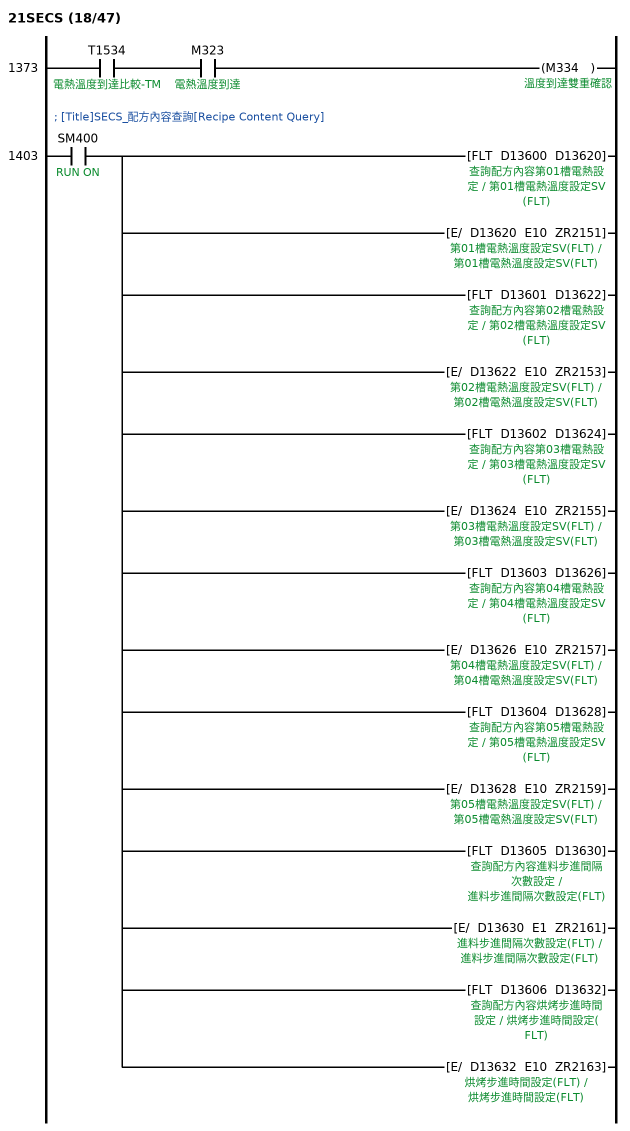
[picture p96: ladder of 21SECS, rungs at steps 1373 to 1403]
1373  LD      T1534  ; 電熱溫度到達比較-TM
      AND     M323  ; 電熱溫度到達
      OUT     M334  ; 溫度到達雙重確認
; [Title]SECS_配方內容查詢[Recipe Content Query]
1403  LD      SM400  ; RUN ON
      FLT     D13600 D13620  ; 查詢配方內容第01槽電熱設定 / 第01槽電熱溫度設定SV(FLT)
      E/      D13620 E10 ZR2151  ; 第01槽電熱溫度設定SV(FLT)
      FLT     D13601 D13622  ; 查詢配方內容第02槽電熱設定 / 第02槽電熱溫度設定SV(FLT)
      E/      D13622 E10 ZR2153  ; 第02槽電熱溫度設定SV(FLT)
      FLT     D13602 D13624  ; 查詢配方內容第03槽電熱設定 / 第03槽電熱溫度設定SV(FLT)
      E/      D13624 E10 ZR2155  ; 第03槽電熱溫度設定SV(FLT)
      FLT     D13603 D13626  ; 查詢配方內容第04槽電熱設定 / 第04槽電熱溫度設定SV(FLT)
      E/      D13626 E10 ZR2157  ; 第04槽電熱溫度設定SV(FLT)
      FLT     D13604 D13628  ; 查詢配方內容第05槽電熱設定 / 第05槽電熱溫度設定SV(FLT)
      E/      D13628 E10 ZR2159  ; 第05槽電熱溫度設定SV(FLT)
      FLT     D13605 D13630  ; 查詢配方內容進料步進間隔次數設定 / 進料步進間隔次數設定(FLT)
      E/      D13630 E1 ZR2161  ; 進料步進間隔次數設定(FLT)
      FLT     D13606 D13632  ; 查詢配方內容烘烤步進時間設定 / 烘烤步進時間設定(FLT)
      E/      D13632 E10 ZR2163  ; 烘烤步進時間設定(FLT)
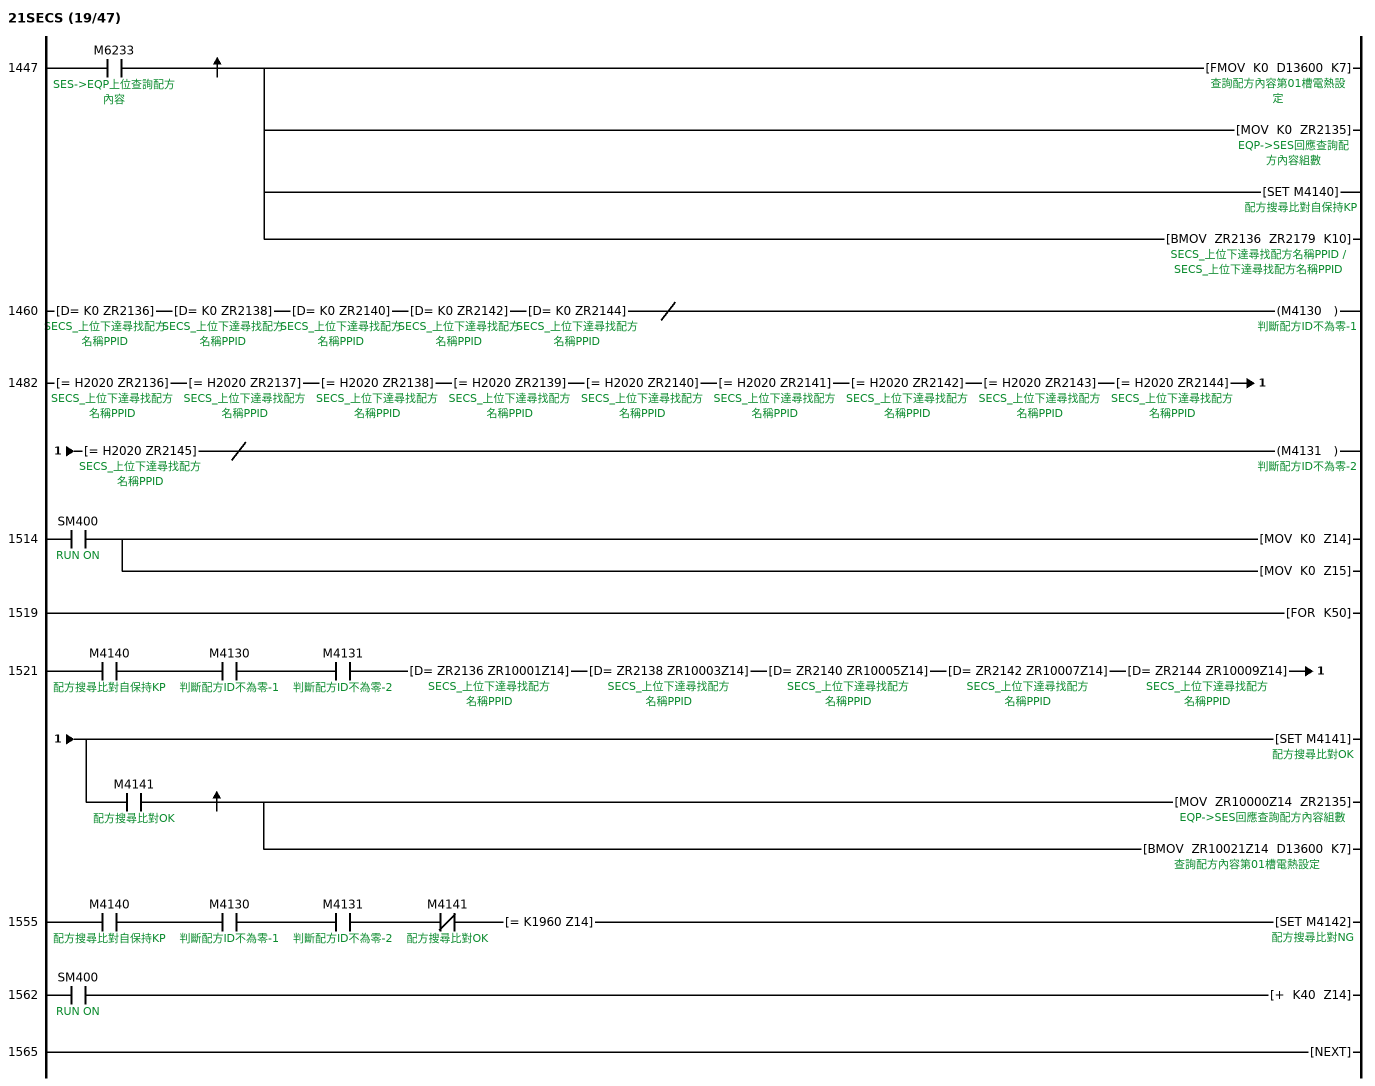
1447  LD      M6233  ; SES->EQP上位查詢配方內容
      MEP
      FMOV    K0 D13600 K7
      MOV     K0 ZR2135  ; EQP->SES回應查詢配方內容組數
      SET     M4140  ; 配方搜尋比對自保持KP
      BMOV    ZR2136 ZR2179 K10  ; SECS_上位下達尋找配方名稱PPID / SECS_上位下達尋找配方名稱PPID
1460  LDD=    K0 ZR2136  ; SECS_上位下達尋找配方名稱PPID
      ANDD=   K0 ZR2138  ; SECS_上位下達尋找配方名稱PPID
      ANDD=   K0 ZR2140  ; SECS_上位下達尋找配方名稱PPID
      ANDD=   K0 ZR2142  ; SECS_上位下達尋找配方名稱PPID
      ANDD=   K0 ZR2144  ; SECS_上位下達尋找配方名稱PPID
      INV
      OUT     M4130  ; 判斷配方ID不為零-1
1482  LD=     H2020 ZR2136  ; SECS_上位下達尋找配方名稱PPID
      AND=    H2020 ZR2137  ; SECS_上位下達尋找配方名稱PPID
      AND=    H2020 ZR2138  ; SECS_上位下達尋找配方名稱PPID
      AND=    H2020 ZR2139  ; SECS_上位下達尋找配方名稱PPID
      AND=    H2020 ZR2140  ; SECS_上位下達尋找配方名稱PPID
      AND=    H2020 ZR2141  ; SECS_上位下達尋找配方名稱PPID
      AND=    H2020 ZR2142  ; SECS_上位下達尋找配方名稱PPID
      AND=    H2020 ZR2143  ; SECS_上位下達尋找配方名稱PPID
      AND=    H2020 ZR2144  ; SECS_上位下達尋找配方名稱PPID
      AND=    H2020 ZR2145  ; SECS_上位下達尋找配方名稱PPID
      INV
      OUT     M4131  ; 判斷配方ID不為零-2
1514  LD      SM400  ; RUN ON
      MOV     K0 Z14
      MOV     K0 Z15
1519  FOR     K50
1521  LD      M4140  ; 配方搜尋比對自保持KP
      AND     M4130  ; 判斷配方ID不為零-1
      AND     M4131  ; 判斷配方ID不為零-2
      ANDD=   ZR2136 ZR10001Z14  ; SECS_上位下達尋找配方名稱PPID
      ANDD=   ZR2138 ZR10003Z14  ; SECS_上位下達尋找配方名稱PPID
      ANDD=   ZR2140 ZR10005Z14  ; SECS_上位下達尋找配方名稱PPID
      ANDD=   ZR2142 ZR10007Z14  ; SECS_上位下達尋找配方名稱PPID
      ANDD=   ZR2144 ZR10009Z14  ; SECS_上位下達尋找配方名稱PPID
      SET     M4141  ; 配方搜尋比對OK
      AND     M4141  ; 配方搜尋比對OK
      MEP
      MOV     ZR10000Z14 ZR2135
      BMOV    ZR10021Z14 D13600 K7
1555  LD      M4140  ; 配方搜尋比對自保持KP
      AND     M4130  ; 判斷配方ID不為零-1
      AND     M4131  ; 判斷配方ID不為零-2
      ANI     M4141  ; 配方搜尋比對OK
      AND=    K1960 Z14
      SET     M4142  ; 配方搜尋比對NG
1562  LD      SM400  ; RUN ON
      +       K40 Z14
1565  NEXT
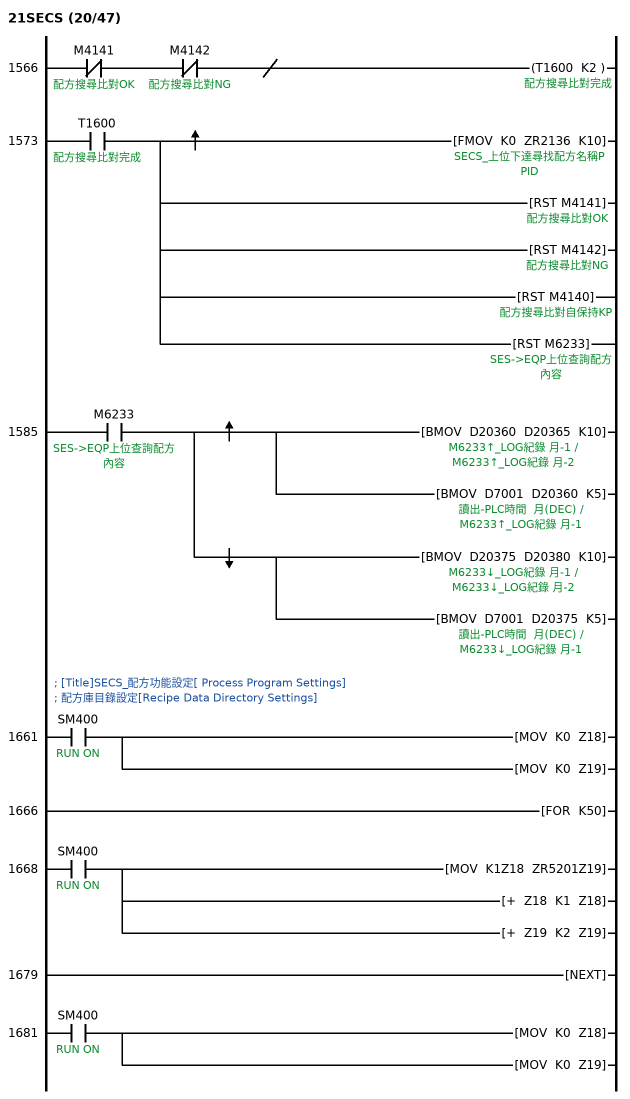
1566  LDI     M4141  ; 配方搜尋比對OK
      ANI     M4142  ; 配方搜尋比對NG
      INV
      OUT     T1600 K2  ; 配方搜尋比對完成
1573  LD      T1600  ; 配方搜尋比對完成
      MPS
      MEP
      FMOV    K0 ZR2136 K10
      MPP
      RST     M4141  ; 配方搜尋比對OK
      RST     M4142  ; 配方搜尋比對NG
      RST     M4140  ; 配方搜尋比對自保持KP
      RST     M6233  ; SES->EQP上位查詢配方內容
1585  LD      M6233  ; SES->EQP上位查詢配方內容
      MPS
      MEP
      BMOV    D20360 D20365 K10  ; M6233↑_LOG紀錄 月-1 / M6233↑_LOG紀錄 月-2
      BMOV    D7001 D20360 K5
      MPP
      MEF
      BMOV    D20375 D20380 K10  ; M6233↓_LOG紀錄 月-1 / M6233↓_LOG紀錄 月-2
      BMOV    D7001 D20375 K5
; [Title]SECS_配方功能設定[ Process Program Settings]
; 配方庫目錄設定[Recipe Data Directory Settings]
1661  LD      SM400  ; RUN ON
      MOV     K0 Z18
      MOV     K0 Z19
1666  FOR     K50
1668  LD      SM400  ; RUN ON
      MOV     K1Z18 ZR5201Z19
      +       Z18 K1 Z18
      +       Z19 K2 Z19
1679  NEXT
1681  LD      SM400  ; RUN ON
      MOV     K0 Z18
      MOV     K0 Z19
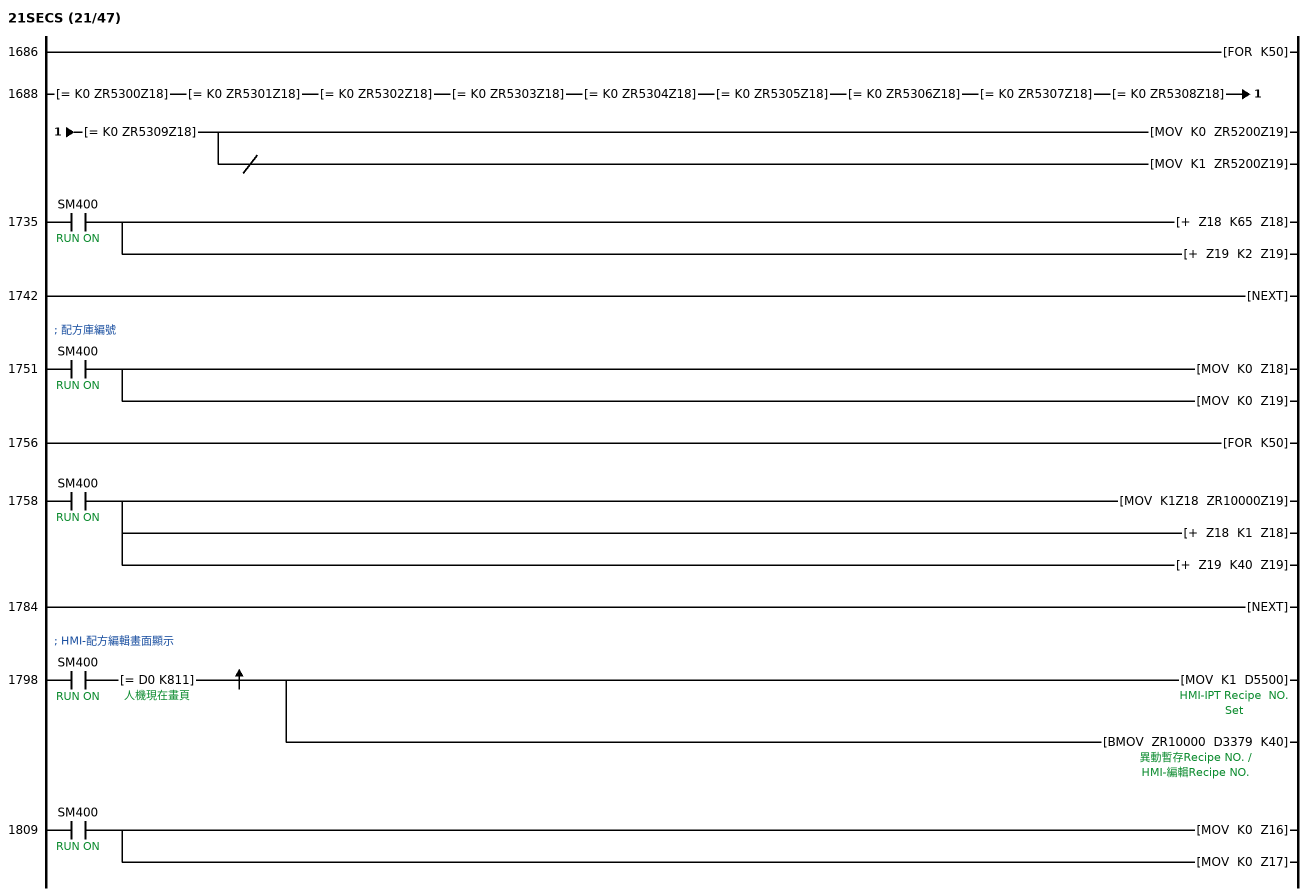
1686  FOR     K50
1688  LD=     K0 ZR5300Z18
      AND=    K0 ZR5301Z18
      AND=    K0 ZR5302Z18
      AND=    K0 ZR5303Z18
      AND=    K0 ZR5304Z18
      AND=    K0 ZR5305Z18
      AND=    K0 ZR5306Z18
      AND=    K0 ZR5307Z18
      AND=    K0 ZR5308Z18
      AND=    K0 ZR5309Z18
      MOV     K0 ZR5200Z19
      INV
      MOV     K1 ZR5200Z19
1735  LD      SM400  ; RUN ON
      +       Z18 K65 Z18
      +       Z19 K2 Z19
1742  NEXT
; 配方庫編號
1751  LD      SM400  ; RUN ON
      MOV     K0 Z18
      MOV     K0 Z19
1756  FOR     K50
1758  LD      SM400  ; RUN ON
      MOV     K1Z18 ZR10000Z19
        [note] 寫入配方參數Recipe NO.編號
      +       Z18 K1 Z18
      +       Z19 K40 Z19
1784  NEXT
; HMI-配方編輯畫面顯示
1798  LD      SM400  ; RUN ON
      AND=    D0 K811  ; 人機現在畫頁
      MEP
      MOV     K1 D5500  ; HMI-IPT Recipe  NO. Set
      BMOV    ZR10000 D3379 K40  ; 異動暫存Recipe NO. / HMI-編輯Recipe NO.
1809  LD      SM400  ; RUN ON
      MOV     K0 Z16
      MOV     K0 Z17
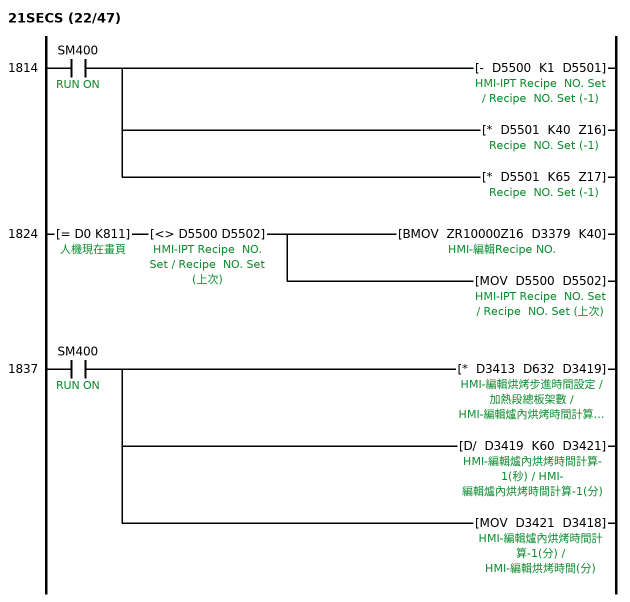
1814  LD      SM400  ; RUN ON
      -       D5500 K1 D5501  ; Recipe  NO. Set (-1)
      *       D5501 K40 Z16
      *       D5501 K65 Z17
1824  LD=     D0 K811  ; 人機現在畫頁
      AND<>   D5500 D5502  ; HMI-IPT Recipe  NO. Set / Recipe  NO. Set (上次)
      BMOV    ZR10000Z16 D3379 K40
      MOV     D5500 D5502
1837  LD      SM400  ; RUN ON
      *       D3413 D632 D3419  ; HMI-編輯烘烤步進時間設定 / 加熱段總板架數 / HMI-編輯爐內烘烤時間計算-1(秒)
        [note] 顯示輸入的秒數換算烘烤時間設定
      D/      D3419 K60 D3421  ; HMI-編輯爐內烘烤時間計算-1(分)
      MOV     D3421 D3418  ; HMI-編輯烘烤時間(分)
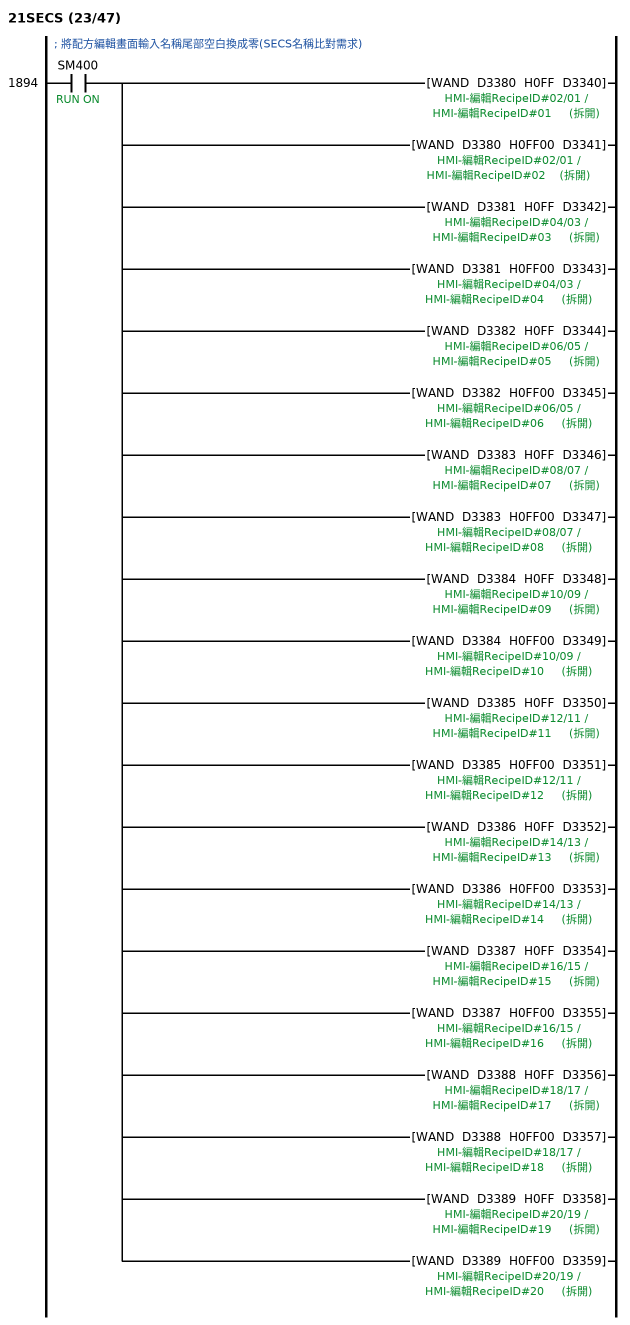
; 將配方編輯畫面輸入名稱尾部空白換成零(SECS名稱比對需求)
1894  LD      SM400  ; RUN ON
      WAND    D3380 H0FF D3340  ; HMI-編輯RecipeID#02/01 / HMI-編輯RecipeID#01     (拆開)
      WAND    D3380 H0FF00 D3341  ; HMI-編輯RecipeID#02    (拆開)
      WAND    D3381 H0FF D3342  ; HMI-編輯RecipeID#04/03 / HMI-編輯RecipeID#03     (拆開)
      WAND    D3381 H0FF00 D3343  ; HMI-編輯RecipeID#04     (拆開)
      WAND    D3382 H0FF D3344  ; HMI-編輯RecipeID#06/05 / HMI-編輯RecipeID#05     (拆開)
      WAND    D3382 H0FF00 D3345  ; HMI-編輯RecipeID#06     (拆開)
      WAND    D3383 H0FF D3346  ; HMI-編輯RecipeID#08/07 / HMI-編輯RecipeID#07     (拆開)
      WAND    D3383 H0FF00 D3347  ; HMI-編輯RecipeID#08     (拆開)
      WAND    D3384 H0FF D3348  ; HMI-編輯RecipeID#10/09 / HMI-編輯RecipeID#09     (拆開)
      WAND    D3384 H0FF00 D3349  ; HMI-編輯RecipeID#10     (拆開)
      WAND    D3385 H0FF D3350  ; HMI-編輯RecipeID#12/11 / HMI-編輯RecipeID#11     (拆開)
      WAND    D3385 H0FF00 D3351  ; HMI-編輯RecipeID#12     (拆開)
      WAND    D3386 H0FF D3352  ; HMI-編輯RecipeID#14/13 / HMI-編輯RecipeID#13     (拆開)
      WAND    D3386 H0FF00 D3353  ; HMI-編輯RecipeID#14     (拆開)
      WAND    D3387 H0FF D3354  ; HMI-編輯RecipeID#16/15 / HMI-編輯RecipeID#15     (拆開)
      WAND    D3387 H0FF00 D3355  ; HMI-編輯RecipeID#16     (拆開)
      WAND    D3388 H0FF D3356  ; HMI-編輯RecipeID#18/17 / HMI-編輯RecipeID#17     (拆開)
      WAND    D3388 H0FF00 D3357  ; HMI-編輯RecipeID#18     (拆開)
      WAND    D3389 H0FF D3358  ; HMI-編輯RecipeID#20/19 / HMI-編輯RecipeID#19     (拆開)
      WAND    D3389 H0FF00 D3359  ; HMI-編輯RecipeID#20     (拆開)
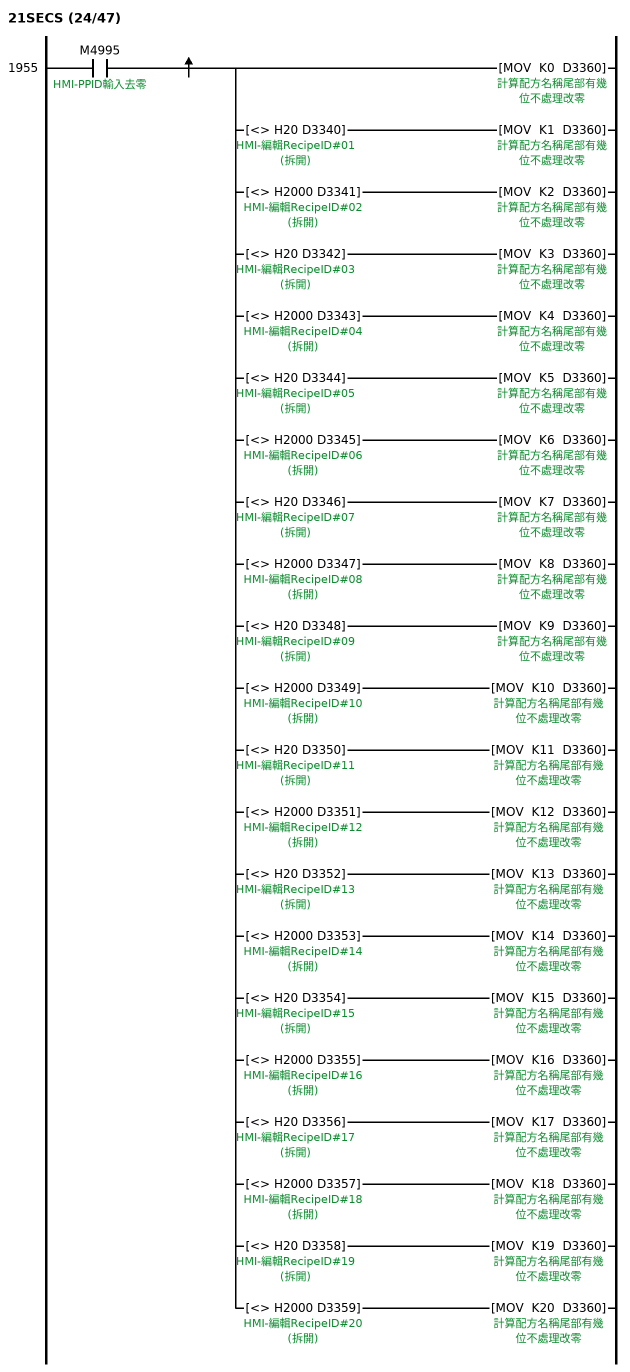
1955  LD      M4995  ; HMI-PPID輸入去零
      MEP
      MOV     K0 D3360  ; 計算配方名稱尾部有幾位不處理改零
      MPS
      AND<>   H20 D3340  ; HMI-編輯RecipeID#01     (拆開)
      MOV     K1 D3360
      MRD
      AND<>   H2000 D3341  ; HMI-編輯RecipeID#02    (拆開)
      MOV     K2 D3360
      MRD
      AND<>   H20 D3342  ; HMI-編輯RecipeID#03     (拆開)
      MOV     K3 D3360
      MRD
      AND<>   H2000 D3343  ; HMI-編輯RecipeID#04     (拆開)
      MOV     K4 D3360
      MRD
      AND<>   H20 D3344  ; HMI-編輯RecipeID#05     (拆開)
      MOV     K5 D3360
      MRD
      AND<>   H2000 D3345  ; HMI-編輯RecipeID#06     (拆開)
      MOV     K6 D3360
      MRD
      AND<>   H20 D3346  ; HMI-編輯RecipeID#07     (拆開)
      MOV     K7 D3360
      MRD
      AND<>   H2000 D3347  ; HMI-編輯RecipeID#08     (拆開)
      MOV     K8 D3360
      MRD
      AND<>   H20 D3348  ; HMI-編輯RecipeID#09     (拆開)
      MOV     K9 D3360
      MRD
      AND<>   H2000 D3349  ; HMI-編輯RecipeID#10     (拆開)
      MOV     K10 D3360
      MRD
      AND<>   H20 D3350  ; HMI-編輯RecipeID#11     (拆開)
      MOV     K11 D3360
      MRD
      AND<>   H2000 D3351  ; HMI-編輯RecipeID#12     (拆開)
      MOV     K12 D3360
      MRD
      AND<>   H20 D3352  ; HMI-編輯RecipeID#13     (拆開)
      MOV     K13 D3360
      MRD
      AND<>   H2000 D3353  ; HMI-編輯RecipeID#14     (拆開)
      MOV     K14 D3360
      MRD
      AND<>   H20 D3354  ; HMI-編輯RecipeID#15     (拆開)
      MOV     K15 D3360
      MRD
      AND<>   H2000 D3355  ; HMI-編輯RecipeID#16     (拆開)
      MOV     K16 D3360
      MRD
      AND<>   H20 D3356  ; HMI-編輯RecipeID#17     (拆開)
      MOV     K17 D3360
      MRD
      AND<>   H2000 D3357  ; HMI-編輯RecipeID#18     (拆開)
      MOV     K18 D3360
      MRD
      AND<>   H20 D3358  ; HMI-編輯RecipeID#19     (拆開)
      MOV     K19 D3360
      MPP
      AND<>   H2000 D3359  ; HMI-編輯RecipeID#20     (拆開)
      MOV     K20 D3360
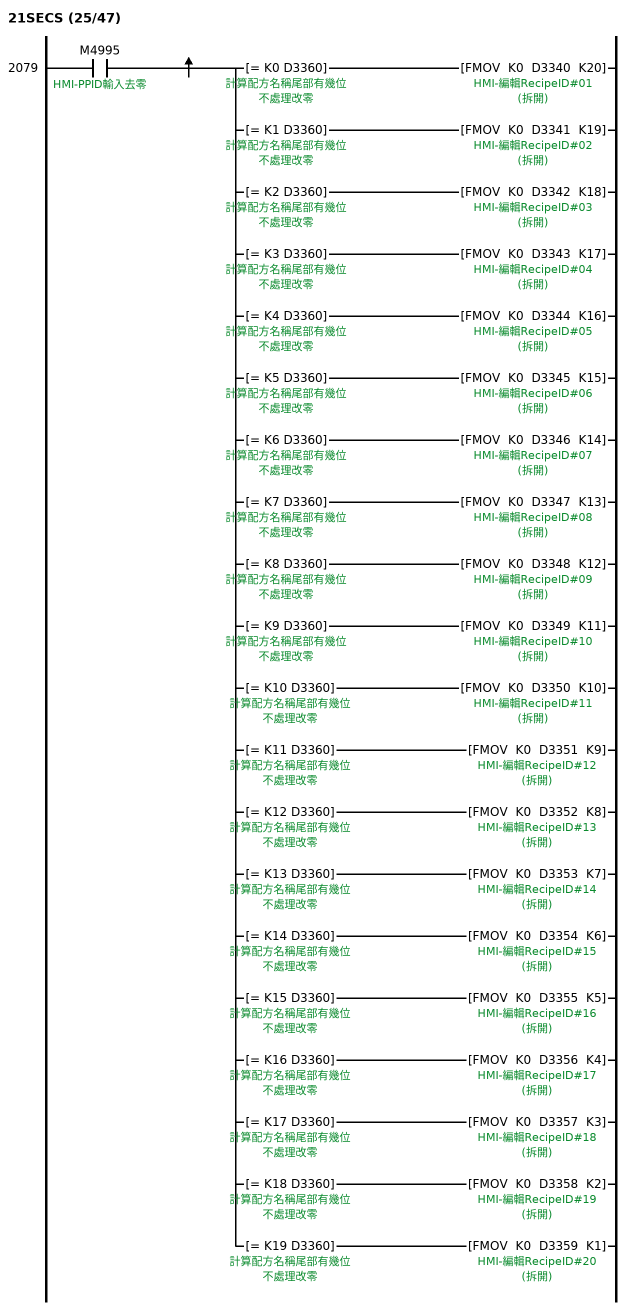
2079  LD      M4995  ; HMI-PPID輸入去零
      MEP
      MPS
      AND=    K0 D3360  ; 計算配方名稱尾部有幾位不處理改零
      FMOV    K0 D3340 K20
      MRD
      AND=    K1 D3360  ; 計算配方名稱尾部有幾位不處理改零
      FMOV    K0 D3341 K19
      MRD
      AND=    K2 D3360  ; 計算配方名稱尾部有幾位不處理改零
      FMOV    K0 D3342 K18
      MRD
      AND=    K3 D3360  ; 計算配方名稱尾部有幾位不處理改零
      FMOV    K0 D3343 K17
      MRD
      AND=    K4 D3360  ; 計算配方名稱尾部有幾位不處理改零
      FMOV    K0 D3344 K16
      MRD
      AND=    K5 D3360  ; 計算配方名稱尾部有幾位不處理改零
      FMOV    K0 D3345 K15
      MRD
      AND=    K6 D3360  ; 計算配方名稱尾部有幾位不處理改零
      FMOV    K0 D3346 K14
      MRD
      AND=    K7 D3360  ; 計算配方名稱尾部有幾位不處理改零
      FMOV    K0 D3347 K13
      MRD
      AND=    K8 D3360  ; 計算配方名稱尾部有幾位不處理改零
      FMOV    K0 D3348 K12
      MRD
      AND=    K9 D3360  ; 計算配方名稱尾部有幾位不處理改零
      FMOV    K0 D3349 K11
      MRD
      AND=    K10 D3360  ; 計算配方名稱尾部有幾位不處理改零
      FMOV    K0 D3350 K10
      MRD
      AND=    K11 D3360  ; 計算配方名稱尾部有幾位不處理改零
      FMOV    K0 D3351 K9
      MRD
      AND=    K12 D3360  ; 計算配方名稱尾部有幾位不處理改零
      FMOV    K0 D3352 K8
      MRD
      AND=    K13 D3360  ; 計算配方名稱尾部有幾位不處理改零
      FMOV    K0 D3353 K7
      MRD
      AND=    K14 D3360  ; 計算配方名稱尾部有幾位不處理改零
      FMOV    K0 D3354 K6
      MRD
      AND=    K15 D3360  ; 計算配方名稱尾部有幾位不處理改零
      FMOV    K0 D3355 K5
      MRD
      AND=    K16 D3360  ; 計算配方名稱尾部有幾位不處理改零
      FMOV    K0 D3356 K4
      MRD
      AND=    K17 D3360  ; 計算配方名稱尾部有幾位不處理改零
      FMOV    K0 D3357 K3
      MRD
      AND=    K18 D3360  ; 計算配方名稱尾部有幾位不處理改零
      FMOV    K0 D3358 K2
      MPP
      AND=    K19 D3360  ; 計算配方名稱尾部有幾位不處理改零
      FMOV    K0 D3359 K1
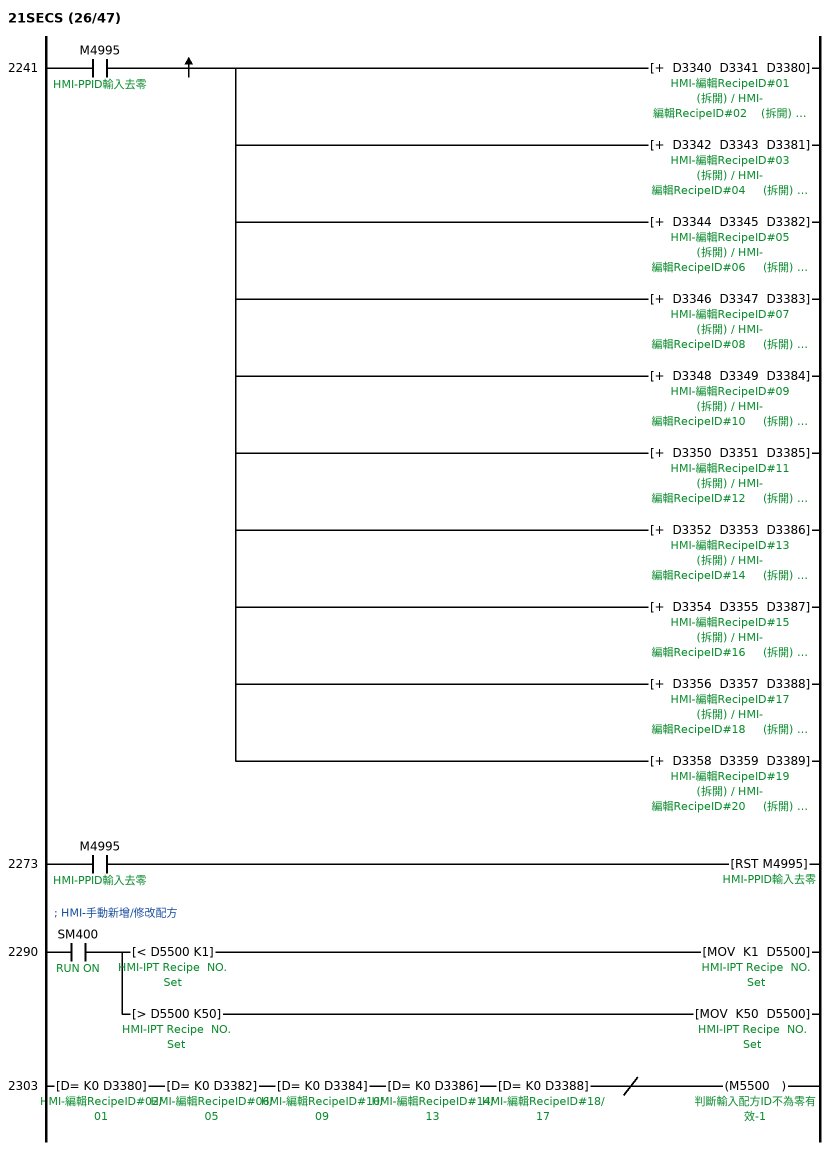
2241  LD      M4995  ; HMI-PPID輸入去零
      MEP
      +       D3340 D3341 D3380
      +       D3342 D3343 D3381
      +       D3344 D3345 D3382
      +       D3346 D3347 D3383
      +       D3348 D3349 D3384
      +       D3350 D3351 D3385
      +       D3352 D3353 D3386
      +       D3354 D3355 D3387
      +       D3356 D3357 D3388
      +       D3358 D3359 D3389
2273  LD      M4995  ; HMI-PPID輸入去零
      RST     M4995  ; HMI-PPID輸入去零
; HMI-手動新增/修改配方
2290  LD      SM400  ; RUN ON
      MPS
      AND<    D5500 K1  ; HMI-IPT Recipe  NO. Set
      MOV     K1 D5500
      MPP
      AND>    D5500 K50  ; HMI-IPT Recipe  NO. Set
      MOV     K50 D5500
2303  LDD=    K0 D3380  ; HMI-編輯RecipeID#02/01
      ANDD=   K0 D3382  ; HMI-編輯RecipeID#06/05
      ANDD=   K0 D3384  ; HMI-編輯RecipeID#10/09
      ANDD=   K0 D3386  ; HMI-編輯RecipeID#14/13
      ANDD=   K0 D3388  ; HMI-編輯RecipeID#18/17
      INV
      OUT     M5500  ; 判斷輸入配方ID不為零有效-1
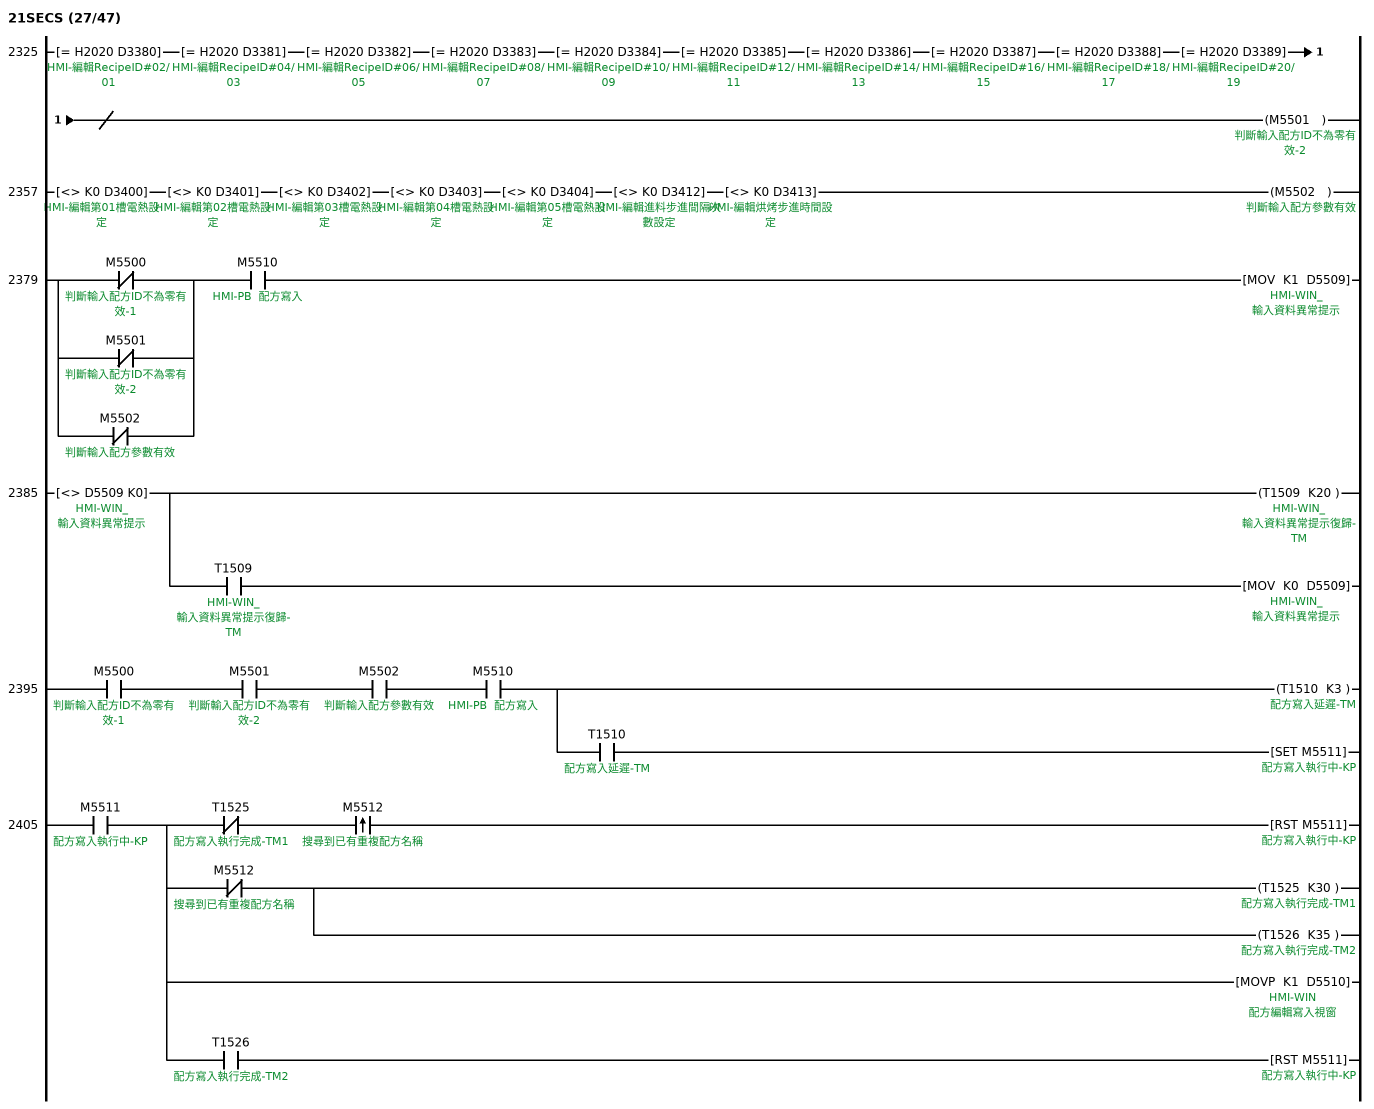
2325  LD=     H2020 D3380  ; HMI-編輯RecipeID#02/01
      AND=    H2020 D3381  ; HMI-編輯RecipeID#04/03
      AND=    H2020 D3382  ; HMI-編輯RecipeID#06/05
      AND=    H2020 D3383  ; HMI-編輯RecipeID#08/07
      AND=    H2020 D3384  ; HMI-編輯RecipeID#10/09
      AND=    H2020 D3385  ; HMI-編輯RecipeID#12/11
      AND=    H2020 D3386  ; HMI-編輯RecipeID#14/13
      AND=    H2020 D3387  ; HMI-編輯RecipeID#16/15
      AND=    H2020 D3388  ; HMI-編輯RecipeID#18/17
      AND=    H2020 D3389  ; HMI-編輯RecipeID#20/19
      INV
      OUT     M5501  ; 判斷輸入配方ID不為零有效-2
2357  LD<>    K0 D3400  ; HMI-編輯第01槽電熱設定
      AND<>   K0 D3401  ; HMI-編輯第02槽電熱設定
      AND<>   K0 D3402  ; HMI-編輯第03槽電熱設定
      AND<>   K0 D3403  ; HMI-編輯第04槽電熱設定
      AND<>   K0 D3404  ; HMI-編輯第05槽電熱設定
      AND<>   K0 D3412  ; HMI-編輯進料步進間隔次數設定
      AND<>   K0 D3413  ; HMI-編輯烘烤步進時間設定
      OUT     M5502  ; 判斷輸入配方參數有效
2379  LDI     M5500  ; 判斷輸入配方ID不為零有效-1
      ORI     M5501  ; 判斷輸入配方ID不為零有效-2
      ORI     M5502  ; 判斷輸入配方參數有效
      AND     M5510  ; HMI-PB  配方寫入
      MOV     K1 D5509  ; HMI-WIN_輸入資料異常提示
2385  LD<>    D5509 K0  ; HMI-WIN_輸入資料異常提示
      OUT     T1509 K20  ; HMI-WIN_輸入資料異常提示復歸-TM
      AND     T1509  ; HMI-WIN_輸入資料異常提示復歸-TM
      MOV     K0 D5509
2395  LD      M5500  ; 判斷輸入配方ID不為零有效-1
      AND     M5501  ; 判斷輸入配方ID不為零有效-2
      AND     M5502  ; 判斷輸入配方參數有效
      AND     M5510  ; HMI-PB  配方寫入
      OUT     T1510 K3  ; 配方寫入延遲-TM
      AND     T1510  ; 配方寫入延遲-TM
      SET     M5511  ; 配方寫入執行中-KP
2405  LD      M5511  ; 配方寫入執行中-KP
      MPS
      ANI     T1525  ; 配方寫入執行完成-TM1
      ANDP    M5512  ; 搜尋到已有重複配方名稱
      RST     M5511  ; 配方寫入執行中-KP
      MRD
      ANI     M5512  ; 搜尋到已有重複配方名稱
      OUT     T1525 K30  ; 配方寫入執行完成-TM1
      OUT     T1526 K35  ; 配方寫入執行完成-TM2
      MPP
      MOVP    K1 D5510  ; HMI-WIN 配方編輯寫入視窗
      AND     T1526  ; 配方寫入執行完成-TM2
      RST     M5511  ; 配方寫入執行中-KP
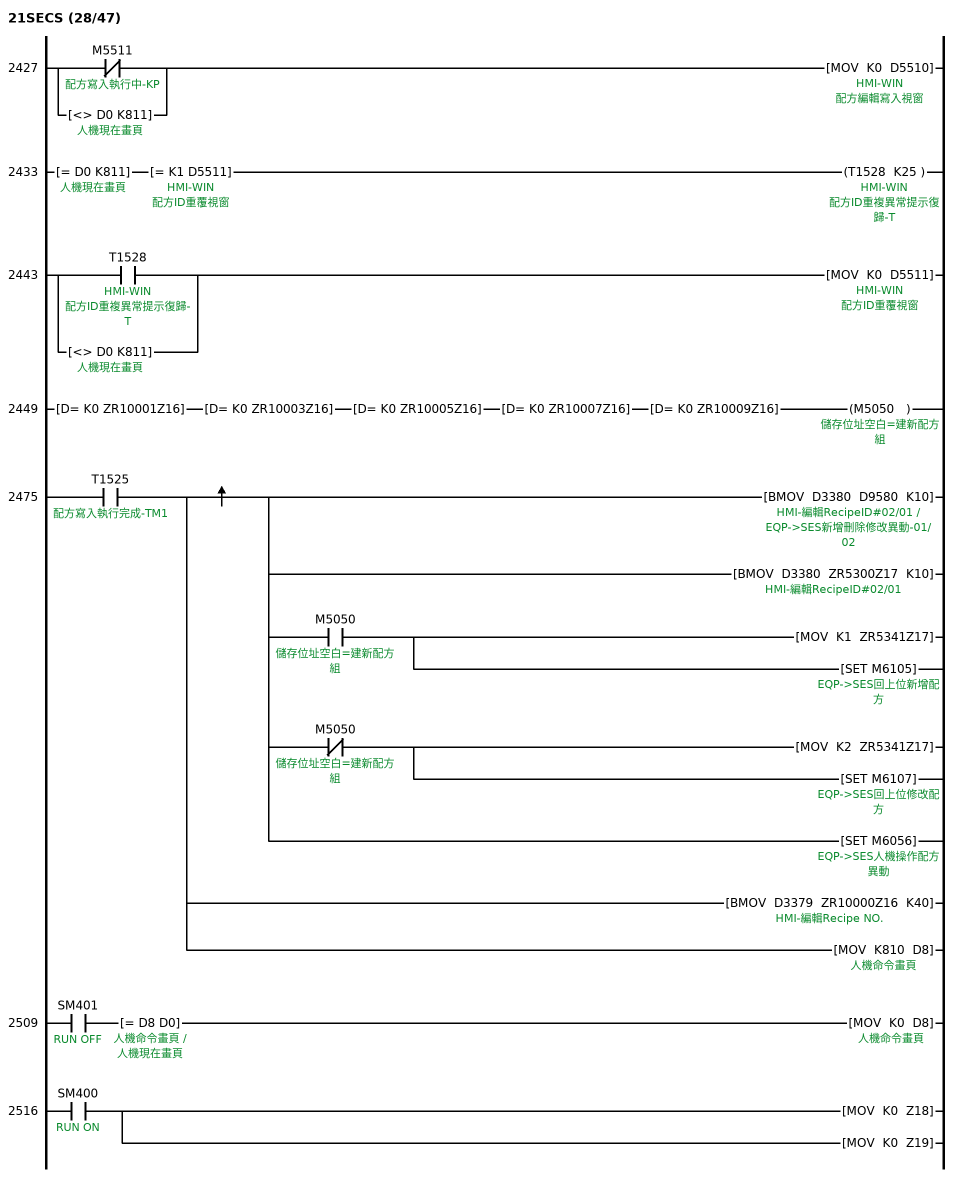
2427  LDI     M5511  ; 配方寫入執行中-KP
      OR<>    D0 K811  ; 人機現在畫頁
      MOV     K0 D5510
2433  LD=     D0 K811  ; 人機現在畫頁
      AND=    K1 D5511  ; HMI-WIN 配方ID重覆視窗
      OUT     T1528 K25  ; HMI-WIN 配方ID重複異常提示復歸-T
2443  LD      T1528  ; HMI-WIN 配方ID重複異常提示復歸-T
      OR<>    D0 K811  ; 人機現在畫頁
      MOV     K0 D5511
2449  LDD=    K0 ZR10001Z16
      ANDD=   K0 ZR10003Z16
      ANDD=   K0 ZR10005Z16
      ANDD=   K0 ZR10007Z16
      ANDD=   K0 ZR10009Z16
      OUT     M5050  ; 儲存位址空白=建新配方組
2475  LD      T1525  ; 配方寫入執行完成-TM1
      MPS
      MEP
      BMOV    D3380 D9580 K10  ; EQP->SES新增刪除修改異動-01/02
      BMOV    D3380 ZR5300Z17 K10
      MPS
      AND     M5050  ; 儲存位址空白=建新配方組
      MOV     K1 ZR5341Z17
      SET     M6105  ; EQP->SES回上位新增配方
      MRD
      ANI     M5050  ; 儲存位址空白=建新配方組
      MOV     K2 ZR5341Z17
      SET     M6107  ; EQP->SES回上位修改配方
      MPP
      SET     M6056  ; EQP->SES人機操作配方異動
      MPP
      BMOV    D3379 ZR10000Z16 K40
      MOV     K810 D8
2509  LD      SM401  ; RUN OFF
      AND=    D8 D0  ; 人機命令畫頁 / 人機現在畫頁
      MOV     K0 D8
2516  LD      SM400  ; RUN ON
      MOV     K0 Z18
      MOV     K0 Z19
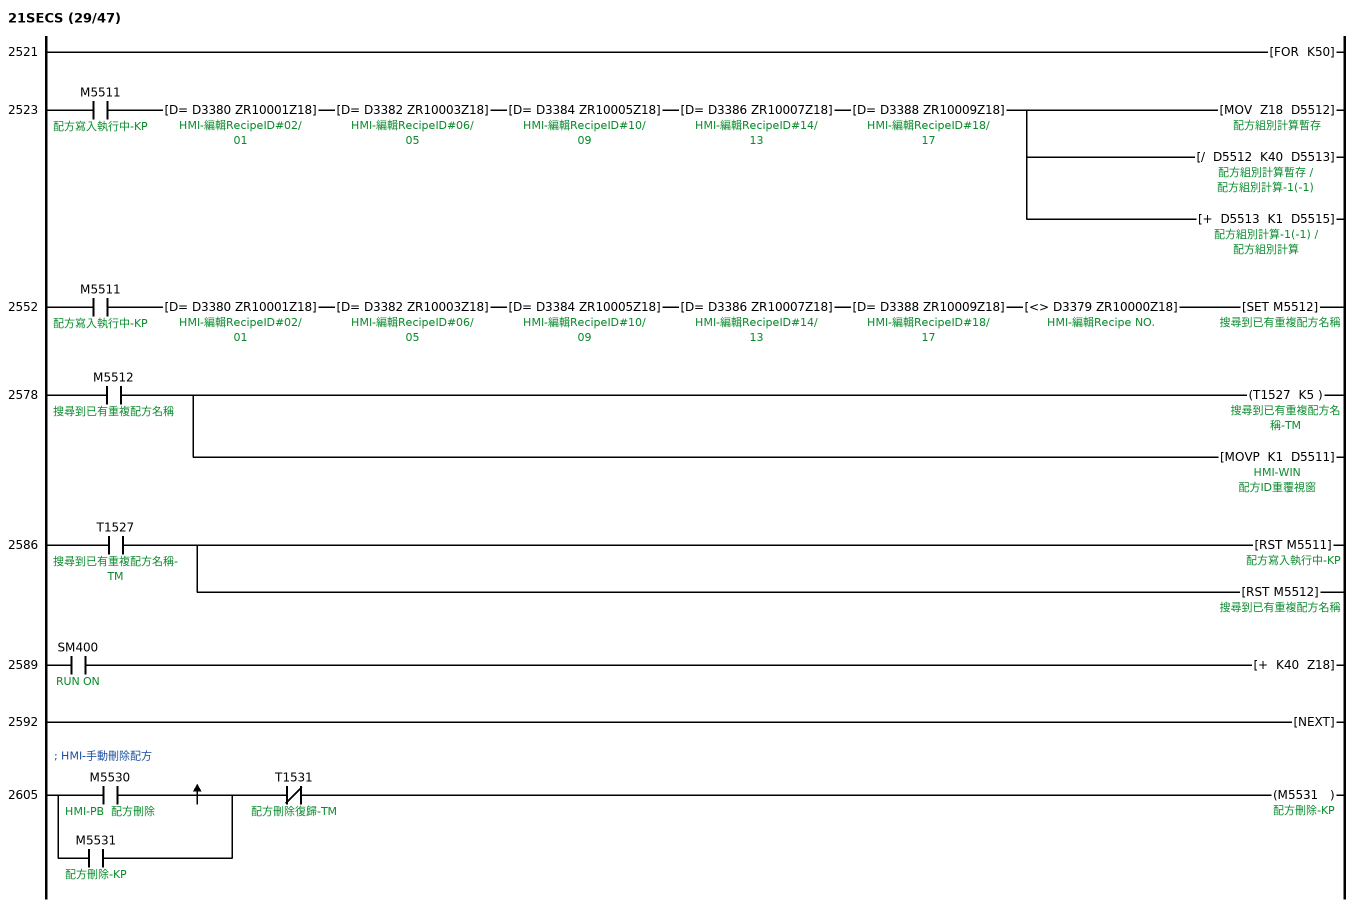
2521  FOR     K50
2523  LD      M5511  ; 配方寫入執行中-KP
      ANDD=   D3380 ZR10001Z18  ; HMI-編輯RecipeID#02/01
      ANDD=   D3382 ZR10003Z18  ; HMI-編輯RecipeID#06/05
      ANDD=   D3384 ZR10005Z18  ; HMI-編輯RecipeID#10/09
      ANDD=   D3386 ZR10007Z18  ; HMI-編輯RecipeID#14/13
      ANDD=   D3388 ZR10009Z18  ; HMI-編輯RecipeID#18/17
      MOV     Z18 D5512  ; 配方組別計算暫存
      /       D5512 K40 D5513  ; 配方組別計算-1(-1)
      +       D5513 K1 D5515  ; 配方組別計算
2552  LD      M5511  ; 配方寫入執行中-KP
      ANDD=   D3380 ZR10001Z18  ; HMI-編輯RecipeID#02/01
      ANDD=   D3382 ZR10003Z18  ; HMI-編輯RecipeID#06/05
      ANDD=   D3384 ZR10005Z18  ; HMI-編輯RecipeID#10/09
      ANDD=   D3386 ZR10007Z18  ; HMI-編輯RecipeID#14/13
      ANDD=   D3388 ZR10009Z18  ; HMI-編輯RecipeID#18/17
      AND<>   D3379 ZR10000Z18  ; HMI-編輯Recipe NO.
      SET     M5512  ; 搜尋到已有重複配方名稱
2578  LD      M5512  ; 搜尋到已有重複配方名稱
      OUT     T1527 K5  ; 搜尋到已有重複配方名稱-TM
      MOVP    K1 D5511
2586  LD      T1527  ; 搜尋到已有重複配方名稱-TM
      RST     M5511  ; 配方寫入執行中-KP
      RST     M5512  ; 搜尋到已有重複配方名稱
2589  LD      SM400  ; RUN ON
      +       K40 Z18
2592  NEXT
; HMI-手動刪除配方
2605  LD      M5530  ; HMI-PB  配方刪除
      MEP
      OR      M5531  ; 配方刪除-KP
      ANI     T1531  ; 配方刪除復歸-TM
      OUT     M5531  ; 配方刪除-KP
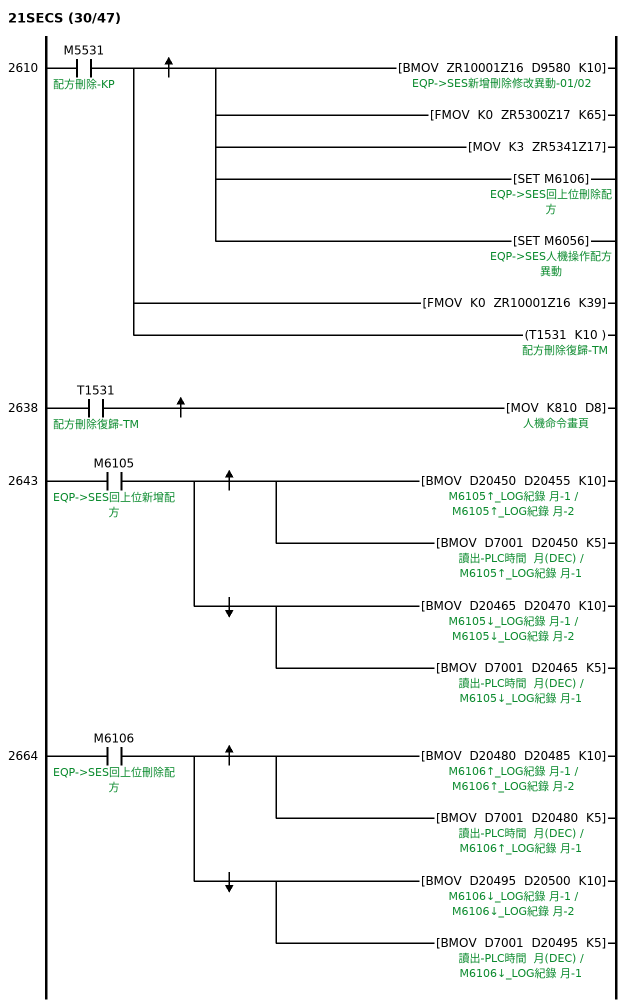
2610  LD      M5531  ; 配方刪除-KP
      MPS
      MEP
      BMOV    ZR10001Z16 D9580 K10
      FMOV    K0 ZR5300Z17 K65
      MOV     K3 ZR5341Z17
      SET     M6106  ; EQP->SES回上位刪除配方
      SET     M6056  ; EQP->SES人機操作配方異動
      MPP
      FMOV    K0 ZR10001Z16 K39
      OUT     T1531 K10  ; 配方刪除復歸-TM
2638  LD      T1531  ; 配方刪除復歸-TM
      MEP
      MOV     K810 D8
2643  LD      M6105  ; EQP->SES回上位新增配方
      MPS
      MEP
      BMOV    D20450 D20455 K10  ; M6105↑_LOG紀錄 月-1 / M6105↑_LOG紀錄 月-2
      BMOV    D7001 D20450 K5
      MPP
      MEF
      BMOV    D20465 D20470 K10  ; M6105↓_LOG紀錄 月-1 / M6105↓_LOG紀錄 月-2
      BMOV    D7001 D20465 K5
2664  LD      M6106  ; EQP->SES回上位刪除配方
      MPS
      MEP
      BMOV    D20480 D20485 K10  ; M6106↑_LOG紀錄 月-1 / M6106↑_LOG紀錄 月-2
      BMOV    D7001 D20480 K5
      MPP
      MEF
      BMOV    D20495 D20500 K10  ; M6106↓_LOG紀錄 月-1 / M6106↓_LOG紀錄 月-2
      BMOV    D7001 D20495 K5
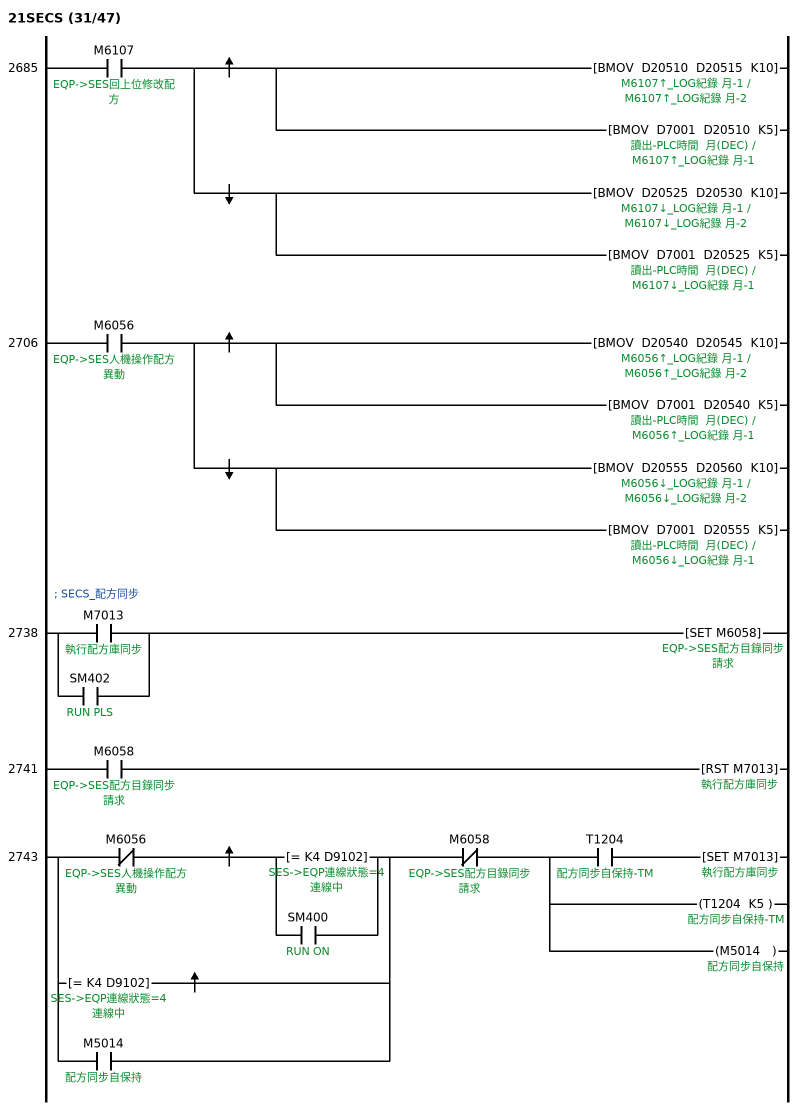
2685  LD      M6107  ; EQP->SES回上位修改配方
      MPS
      MEP
      BMOV    D20510 D20515 K10  ; M6107↑_LOG紀錄 月-1 / M6107↑_LOG紀錄 月-2
      BMOV    D7001 D20510 K5
      MPP
      MEF
      BMOV    D20525 D20530 K10  ; M6107↓_LOG紀錄 月-1 / M6107↓_LOG紀錄 月-2
      BMOV    D7001 D20525 K5
2706  LD      M6056  ; EQP->SES人機操作配方異動
      MPS
      MEP
      BMOV    D20540 D20545 K10  ; M6056↑_LOG紀錄 月-1 / M6056↑_LOG紀錄 月-2
      BMOV    D7001 D20540 K5
      MPP
      MEF
      BMOV    D20555 D20560 K10  ; M6056↓_LOG紀錄 月-1 / M6056↓_LOG紀錄 月-2
      BMOV    D7001 D20555 K5
; SECS_配方同步
2738  LD      M7013  ; 執行配方庫同步
      OR      SM402  ; RUN PLS
      SET     M6058  ; EQP->SES配方目錄同步請求
2741  LD      M6058  ; EQP->SES配方目錄同步請求
      RST     M7013  ; 執行配方庫同步
2743  LDI     M6056  ; EQP->SES人機操作配方異動
      MEP
      LD=     K4 D9102  ; SES->EQP連線狀態=4      連線中
      OR      SM400  ; RUN ON
      ANB
      LD=     K4 D9102  ; SES->EQP連線狀態=4      連線中
      MEP
      ORB
      OR      M5014  ; 配方同步自保持
      ANI     M6058  ; EQP->SES配方目錄同步請求
      MPS
      AND     T1204  ; 配方同步自保持-TM
      SET     M7013  ; 執行配方庫同步
      MPP
      OUT     T1204 K5  ; 配方同步自保持-TM
      OUT     M5014  ; 配方同步自保持
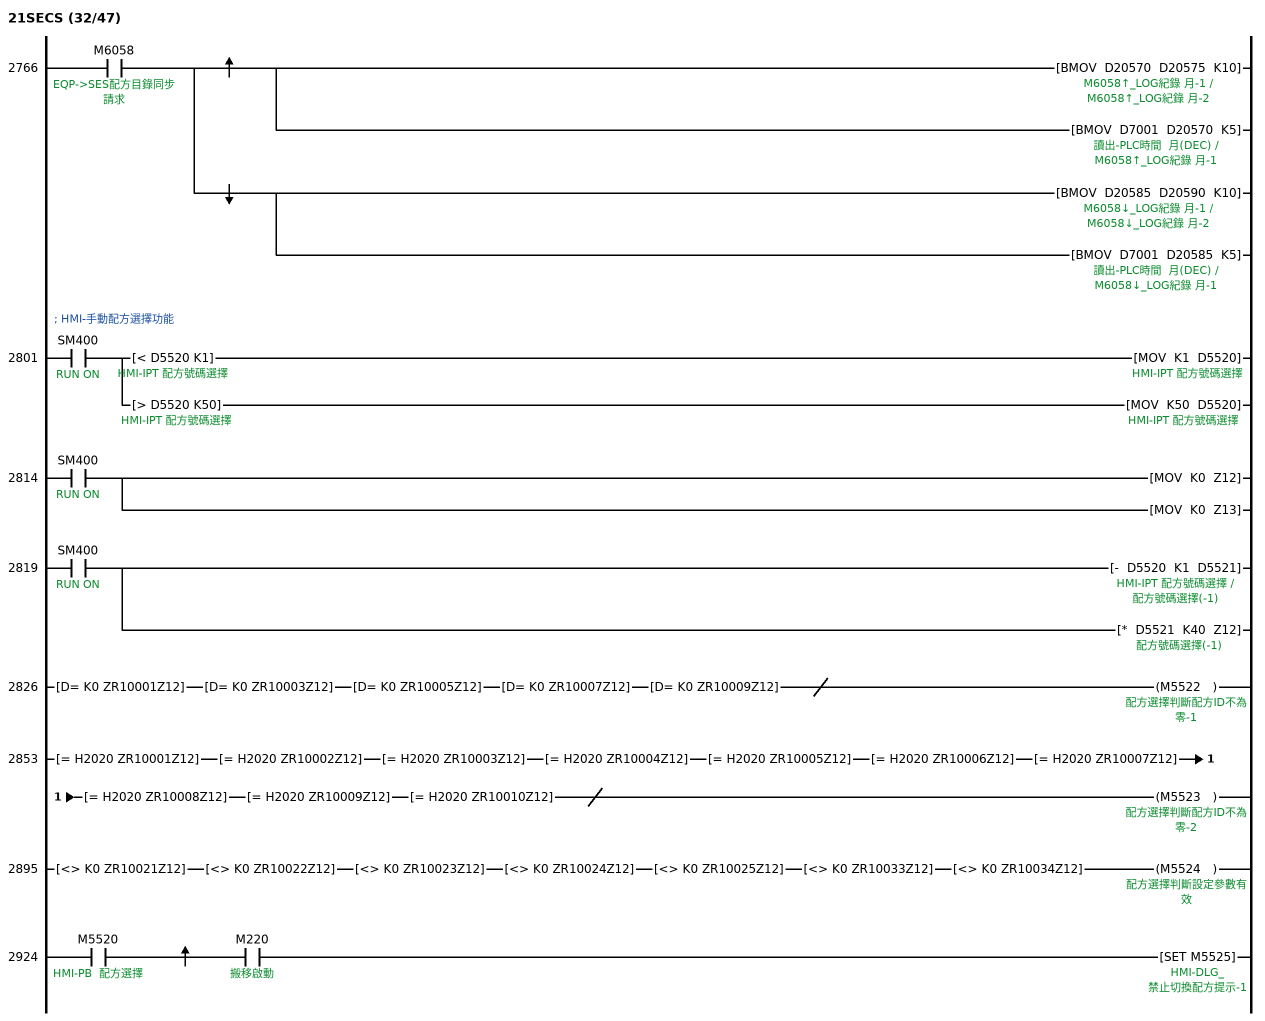
2766  LD      M6058  ; EQP->SES配方目錄同步請求
      MPS
      MEP
      BMOV    D20570 D20575 K10  ; M6058↑_LOG紀錄 月-1 / M6058↑_LOG紀錄 月-2
      BMOV    D7001 D20570 K5
      MPP
      MEF
      BMOV    D20585 D20590 K10  ; M6058↓_LOG紀錄 月-1 / M6058↓_LOG紀錄 月-2
      BMOV    D7001 D20585 K5
; HMI-手動配方選擇功能
2801  LD      SM400  ; RUN ON
      MPS
      AND<    D5520 K1  ; HMI-IPT 配方號碼選擇
      MOV     K1 D5520
      MPP
      AND>    D5520 K50  ; HMI-IPT 配方號碼選擇
      MOV     K50 D5520
2814  LD      SM400  ; RUN ON
      MOV     K0 Z12
      MOV     K0 Z13
2819  LD      SM400  ; RUN ON
      -       D5520 K1 D5521  ; 配方號碼選擇(-1)
      *       D5521 K40 Z12
2826  LDD=    K0 ZR10001Z12
      ANDD=   K0 ZR10003Z12
      ANDD=   K0 ZR10005Z12
      ANDD=   K0 ZR10007Z12
      ANDD=   K0 ZR10009Z12
      INV
      OUT     M5522  ; 配方選擇判斷配方ID不為零-1
2853  LD=     H2020 ZR10001Z12
      AND=    H2020 ZR10002Z12
      AND=    H2020 ZR10003Z12
      AND=    H2020 ZR10004Z12
      AND=    H2020 ZR10005Z12
      AND=    H2020 ZR10006Z12
      AND=    H2020 ZR10007Z12
      AND=    H2020 ZR10008Z12
      AND=    H2020 ZR10009Z12
      AND=    H2020 ZR10010Z12
      INV
      OUT     M5523  ; 配方選擇判斷配方ID不為零-2
2895  LD<>    K0 ZR10021Z12
      AND<>   K0 ZR10022Z12
      AND<>   K0 ZR10023Z12
      AND<>   K0 ZR10024Z12
      AND<>   K0 ZR10025Z12
      AND<>   K0 ZR10033Z12
      AND<>   K0 ZR10034Z12
      OUT     M5524  ; 配方選擇判斷設定參數有效
2924  LD      M5520  ; HMI-PB  配方選擇
      MEP
      AND     M220  ; 搬移啟動
      SET     M5525  ; HMI-DLG_禁止切換配方提示-1
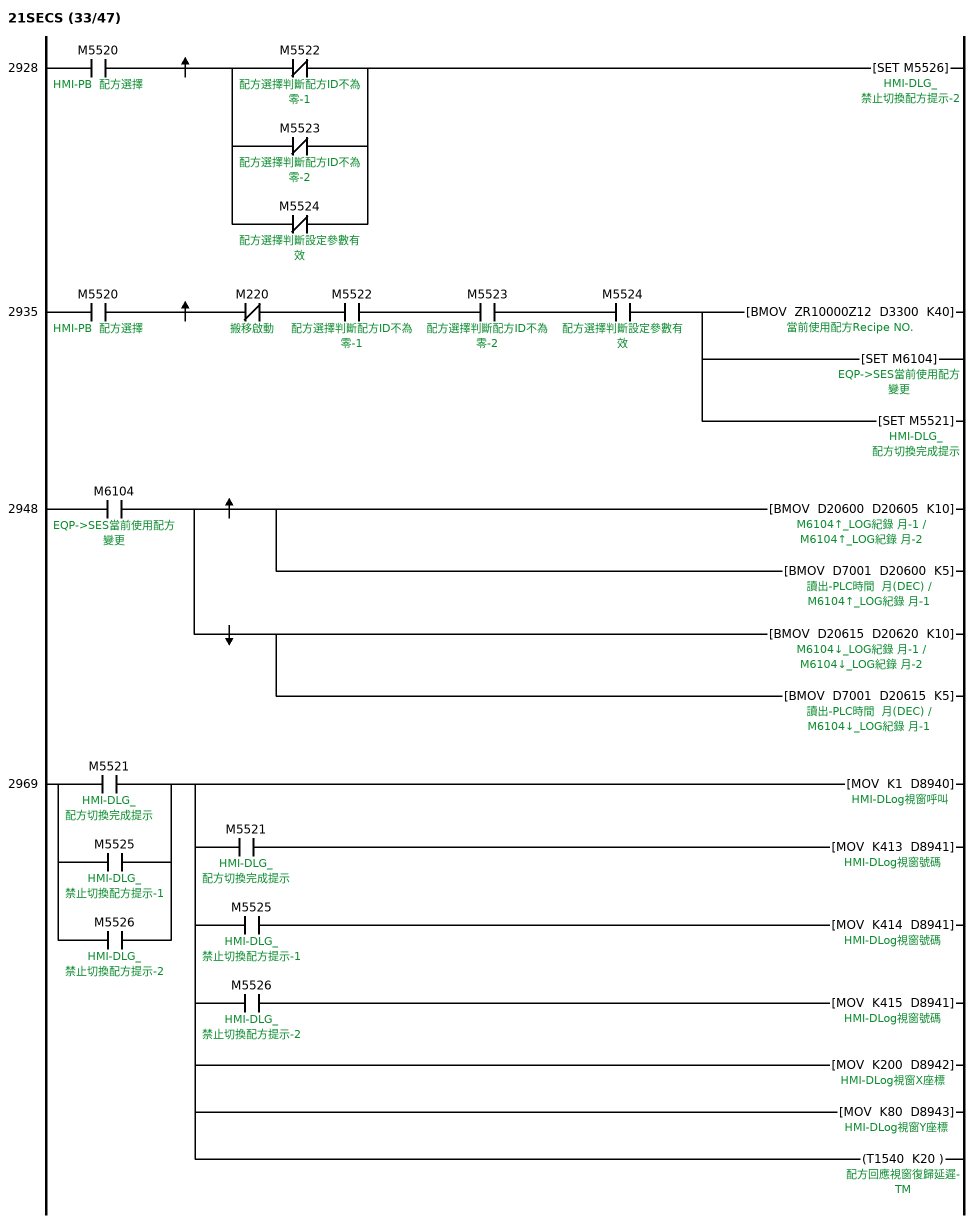
2928  LD      M5520  ; HMI-PB  配方選擇
      MEP
      LDI     M5522  ; 配方選擇判斷配方ID不為零-1
      ORI     M5523  ; 配方選擇判斷配方ID不為零-2
      ORI     M5524  ; 配方選擇判斷設定參數有效
      ANB
      SET     M5526  ; HMI-DLG_禁止切換配方提示-2
2935  LD      M5520  ; HMI-PB  配方選擇
      MEP
      ANI     M220  ; 搬移啟動
      AND     M5522  ; 配方選擇判斷配方ID不為零-1
      AND     M5523  ; 配方選擇判斷配方ID不為零-2
      AND     M5524  ; 配方選擇判斷設定參數有效
      BMOV    ZR10000Z12 D3300 K40  ; 當前使用配方Recipe NO.
      SET     M6104  ; EQP->SES當前使用配方變更
      SET     M5521  ; HMI-DLG_配方切換完成提示
2948  LD      M6104  ; EQP->SES當前使用配方變更
      MPS
      MEP
      BMOV    D20600 D20605 K10  ; M6104↑_LOG紀錄 月-1 / M6104↑_LOG紀錄 月-2
      BMOV    D7001 D20600 K5
      MPP
      MEF
      BMOV    D20615 D20620 K10  ; M6104↓_LOG紀錄 月-1 / M6104↓_LOG紀錄 月-2
      BMOV    D7001 D20615 K5
2969  LD      M5521  ; HMI-DLG_配方切換完成提示
      OR      M5525  ; HMI-DLG_禁止切換配方提示-1
      OR      M5526  ; HMI-DLG_禁止切換配方提示-2
      MOV     K1 D8940  ; HMI-DLog視窗呼叫
      MPS
      AND     M5521  ; HMI-DLG_配方切換完成提示
      MOV     K413 D8941  ; HMI-DLog視窗號碼
      MRD
      AND     M5525  ; HMI-DLG_禁止切換配方提示-1
      MOV     K414 D8941
      MRD
      AND     M5526  ; HMI-DLG_禁止切換配方提示-2
      MOV     K415 D8941
      MPP
      MOV     K200 D8942  ; HMI-DLog視窗X座標
      MOV     K80 D8943  ; HMI-DLog視窗Y座標
      OUT     T1540 K20  ; 配方回應視窗復歸延遲-TM
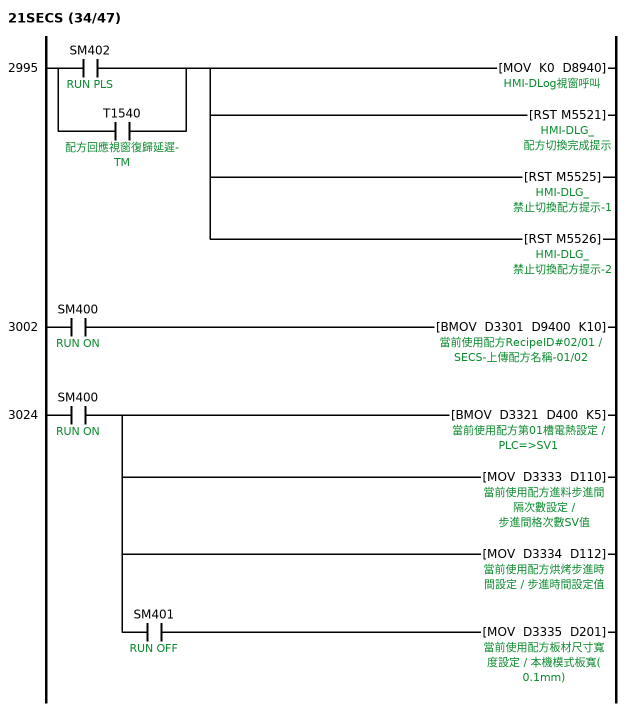
2995  LD      SM402  ; RUN PLS
      OR      T1540  ; 配方回應視窗復歸延遲-TM
      MOV     K0 D8940
      RST     M5521  ; HMI-DLG_配方切換完成提示
      RST     M5525  ; HMI-DLG_禁止切換配方提示-1
      RST     M5526  ; HMI-DLG_禁止切換配方提示-2
3002  LD      SM400  ; RUN ON
      BMOV    D3301 D9400 K10  ; 當前使用配方RecipeID#02/01 / SECS-上傳配方名稱-01/02
        [note] D9400_上報SECS目前使用PPID名稱
3024  LD      SM400  ; RUN ON
      BMOV    D3321 D400 K5  ; 當前使用配方第01槽電熱設定
      MOV     D3333 D110  ; 當前使用配方進料步進間隔次數設定
      MOV     D3334 D112  ; 當前使用配方烘烤步進時間設定
      AND     SM401  ; RUN OFF
      MOV     D3335 D201  ; 當前使用配方板材尺寸寬度設定
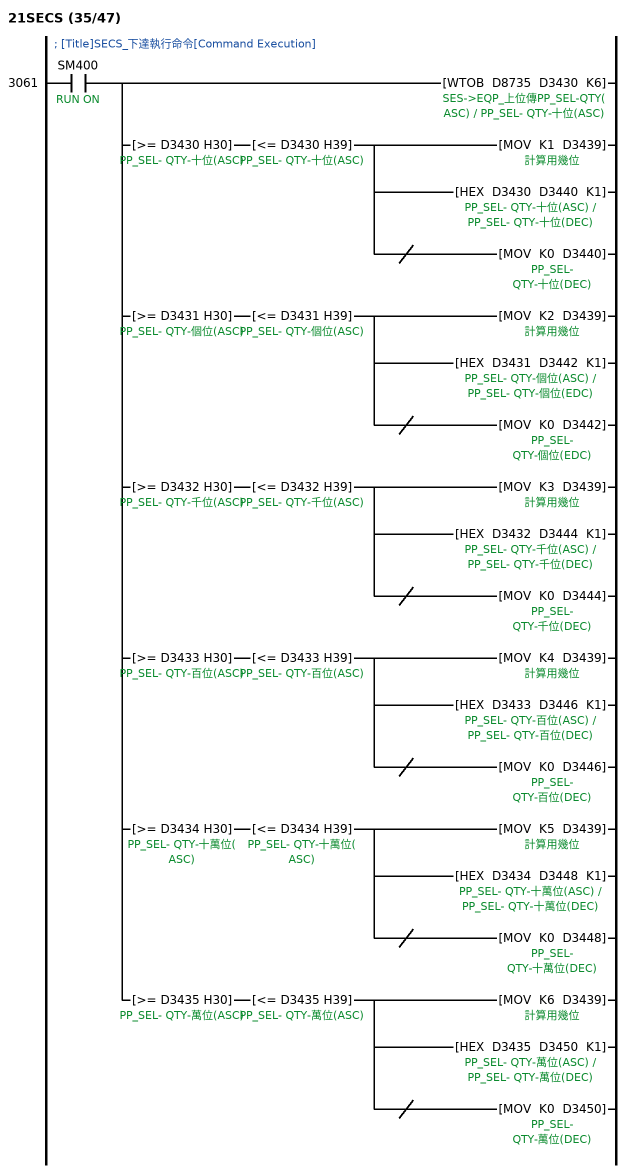
; [Title]SECS_下達執行命令[Command Execution]
3061  LD      SM400  ; RUN ON
      WTOB    D8735 D3430 K6  ; SES->EQP_上位傳PP_SEL-QTY(ASC) / PP_SEL- QTY-十位(ASC)
      MPS
      AND>=   D3430 H30  ; PP_SEL- QTY-十位(ASC)
      AND<=   D3430 H39  ; PP_SEL- QTY-十位(ASC)
      MOV     K1 D3439  ; 計算用幾位
      HEX     D3430 D3440 K1  ; PP_SEL- QTY-十位(DEC)
      INV
      MOV     K0 D3440
      MRD
      AND>=   D3431 H30  ; PP_SEL- QTY-個位(ASC)
      AND<=   D3431 H39  ; PP_SEL- QTY-個位(ASC)
      MOV     K2 D3439
      HEX     D3431 D3442 K1  ; PP_SEL- QTY-個位(EDC)
      INV
      MOV     K0 D3442
      MRD
      AND>=   D3432 H30  ; PP_SEL- QTY-千位(ASC)
      AND<=   D3432 H39  ; PP_SEL- QTY-千位(ASC)
      MOV     K3 D3439
      HEX     D3432 D3444 K1  ; PP_SEL- QTY-千位(DEC)
      INV
      MOV     K0 D3444
      MRD
      AND>=   D3433 H30  ; PP_SEL- QTY-百位(ASC)
      AND<=   D3433 H39  ; PP_SEL- QTY-百位(ASC)
      MOV     K4 D3439
      HEX     D3433 D3446 K1  ; PP_SEL- QTY-百位(DEC)
      INV
      MOV     K0 D3446
      MRD
      AND>=   D3434 H30  ; PP_SEL- QTY-十萬位(ASC)
      AND<=   D3434 H39  ; PP_SEL- QTY-十萬位(ASC)
      MOV     K5 D3439
      HEX     D3434 D3448 K1  ; PP_SEL- QTY-十萬位(DEC)
      INV
      MOV     K0 D3448
      MPP
      AND>=   D3435 H30  ; PP_SEL- QTY-萬位(ASC)
      AND<=   D3435 H39  ; PP_SEL- QTY-萬位(ASC)
      MOV     K6 D3439
      HEX     D3435 D3450 K1  ; PP_SEL- QTY-萬位(DEC)
      INV
      MOV     K0 D3450
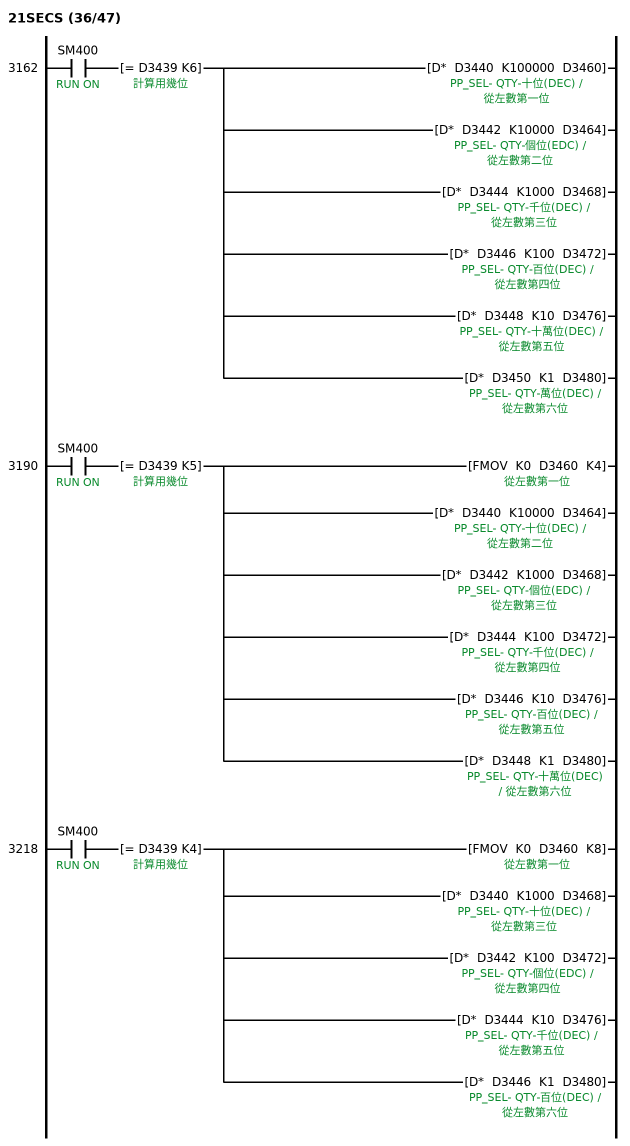
3162  LD      SM400  ; RUN ON
      AND=    D3439 K6  ; 計算用幾位
      D*      D3440 K100000 D3460  ; 從左數第一位
      D*      D3442 K10000 D3464  ; 從左數第二位
      D*      D3444 K1000 D3468  ; 從左數第三位
      D*      D3446 K100 D3472  ; 從左數第四位
      D*      D3448 K10 D3476  ; 從左數第五位
      D*      D3450 K1 D3480  ; 從左數第六位
3190  LD      SM400  ; RUN ON
      AND=    D3439 K5  ; 計算用幾位
      FMOV    K0 D3460 K4
      D*      D3440 K10000 D3464
      D*      D3442 K1000 D3468
      D*      D3444 K100 D3472
      D*      D3446 K10 D3476
      D*      D3448 K1 D3480
3218  LD      SM400  ; RUN ON
      AND=    D3439 K4  ; 計算用幾位
      FMOV    K0 D3460 K8
      D*      D3440 K1000 D3468
      D*      D3442 K100 D3472
      D*      D3444 K10 D3476
      D*      D3446 K1 D3480
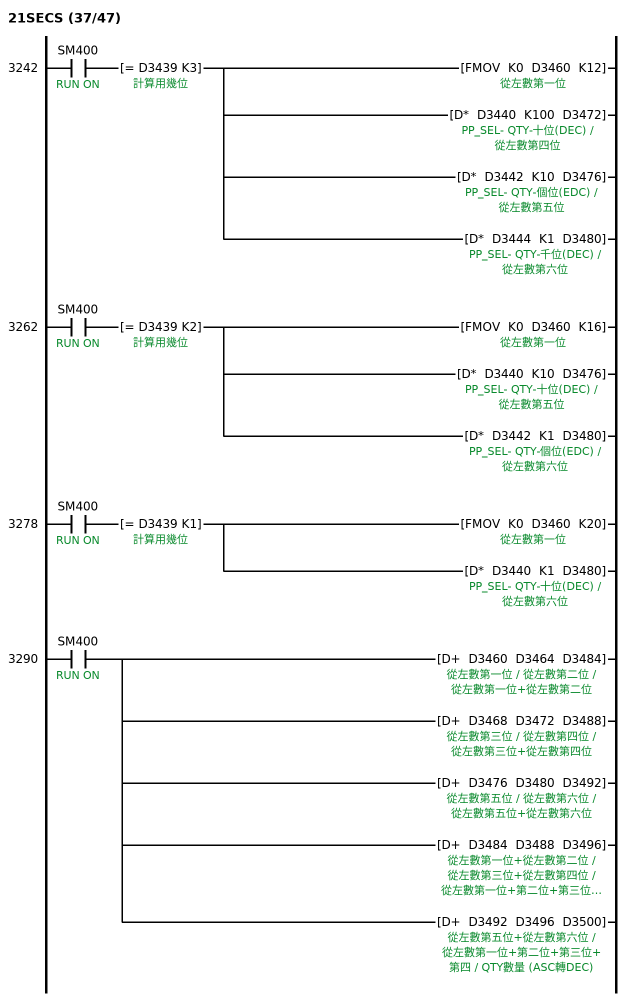
3242  LD      SM400  ; RUN ON
      AND=    D3439 K3  ; 計算用幾位
      FMOV    K0 D3460 K12
      D*      D3440 K100 D3472
      D*      D3442 K10 D3476
      D*      D3444 K1 D3480
3262  LD      SM400  ; RUN ON
      AND=    D3439 K2  ; 計算用幾位
      FMOV    K0 D3460 K16
      D*      D3440 K10 D3476
      D*      D3442 K1 D3480
3278  LD      SM400  ; RUN ON
      AND=    D3439 K1  ; 計算用幾位
      FMOV    K0 D3460 K20
      D*      D3440 K1 D3480
3290  LD      SM400  ; RUN ON
      D+      D3460 D3464 D3484  ; 從左數第一位+從左數第二位
      D+      D3468 D3472 D3488  ; 從左數第三位+從左數第四位
      D+      D3476 D3480 D3492  ; 從左數第五位+從左數第六位
      D+      D3484 D3488 D3496  ; 從左數第一位+第二位+第三位+第四
      D+      D3492 D3496 D3500  ; QTY數量 (ASC轉DEC)
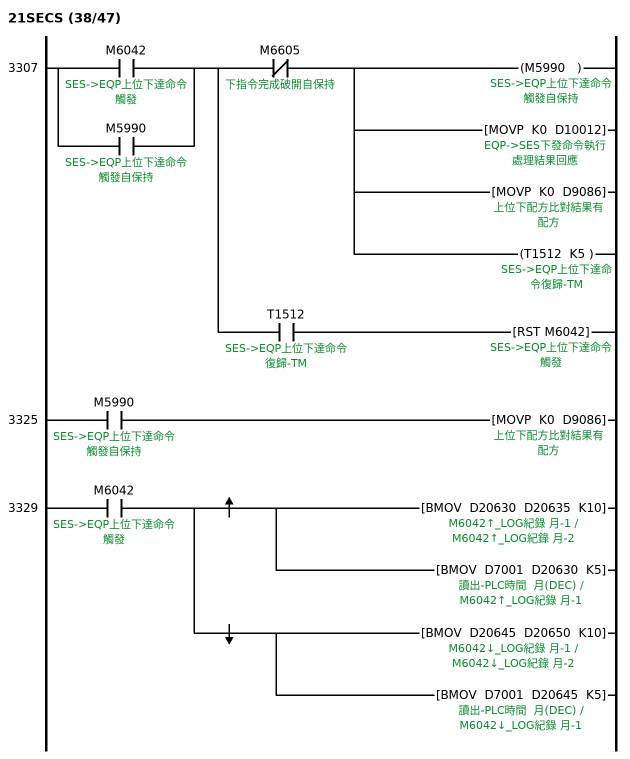
3307  LD      M6042  ; SES->EQP上位下達命令觸發
      OR      M5990  ; SES->EQP上位下達命令觸發自保持
      MPS
      ANI     M6605  ; 下指令完成破開自保持
      OUT     M5990  ; SES->EQP上位下達命令觸發自保持
      MOVP    K0 D10012  ; EQP->SES下發命令執行處理結果回應
      MOVP    K0 D9086  ; 上位下配方比對結果有配方
      OUT     T1512 K5  ; SES->EQP上位下達命令復歸-TM
      MPP
      AND     T1512  ; SES->EQP上位下達命令復歸-TM
      RST     M6042  ; SES->EQP上位下達命令觸發
3325  LD      M5990  ; SES->EQP上位下達命令觸發自保持
      MOVP    K0 D9086
3329  LD      M6042  ; SES->EQP上位下達命令觸發
      MPS
      MEP
      BMOV    D20630 D20635 K10  ; M6042↑_LOG紀錄 月-1 / M6042↑_LOG紀錄 月-2
      BMOV    D7001 D20630 K5
      MPP
      MEF
      BMOV    D20645 D20650 K10  ; M6042↓_LOG紀錄 月-1 / M6042↓_LOG紀錄 月-2
      BMOV    D7001 D20645 K5
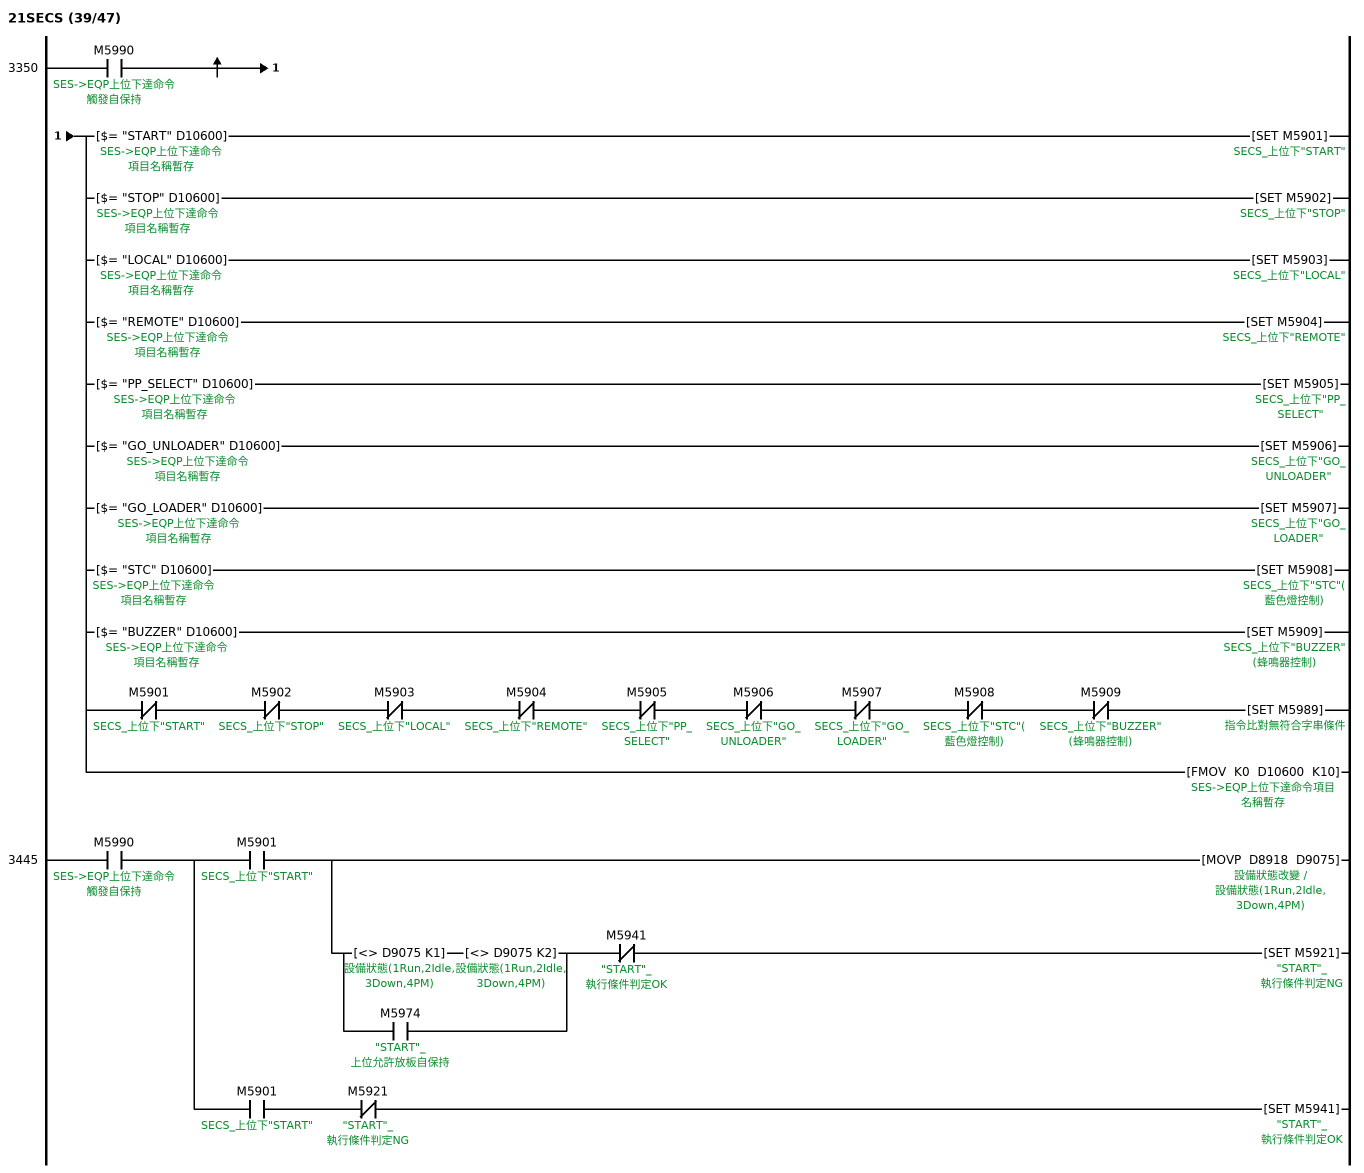
3350  LD      M5990  ; SES->EQP上位下達命令觸發自保持
      MEP
      MPS
      AND$=   "START" D10600  ; SES->EQP上位下達命令項目名稱暫存
      SET     M5901  ; SECS_上位下"START"
      MRD
      AND$=   "STOP" D10600  ; SES->EQP上位下達命令項目名稱暫存
      SET     M5902  ; SECS_上位下"STOP"
      MRD
      AND$=   "LOCAL" D10600  ; SES->EQP上位下達命令項目名稱暫存
      SET     M5903  ; SECS_上位下"LOCAL"
      MRD
      AND$=   "REMOTE" D10600  ; SES->EQP上位下達命令項目名稱暫存
      SET     M5904  ; SECS_上位下"REMOTE"
      MRD
      AND$=   "PP_SELECT" D10600  ; SES->EQP上位下達命令項目名稱暫存
      SET     M5905  ; SECS_上位下"PP_SELECT"
      MRD
      AND$=   "GO_UNLOADER" D10600  ; SES->EQP上位下達命令項目名稱暫存
      SET     M5906  ; SECS_上位下"GO_UNLOADER"
      MRD
      AND$=   "GO_LOADER" D10600  ; SES->EQP上位下達命令項目名稱暫存
      SET     M5907  ; SECS_上位下"GO_LOADER"
      MRD
      AND$=   "STC" D10600  ; SES->EQP上位下達命令項目名稱暫存
      SET     M5908  ; SECS_上位下"STC"(藍色燈控制)
      MRD
      AND$=   "BUZZER" D10600  ; SES->EQP上位下達命令項目名稱暫存
      SET     M5909  ; SECS_上位下"BUZZER"(蜂鳴器控制)
      MRD
      ANI     M5901  ; SECS_上位下"START"
      ANI     M5902  ; SECS_上位下"STOP"
      ANI     M5903  ; SECS_上位下"LOCAL"
      ANI     M5904  ; SECS_上位下"REMOTE"
      ANI     M5905  ; SECS_上位下"PP_SELECT"
      ANI     M5906  ; SECS_上位下"GO_UNLOADER"
      ANI     M5907  ; SECS_上位下"GO_LOADER"
      ANI     M5908  ; SECS_上位下"STC"(藍色燈控制)
      ANI     M5909  ; SECS_上位下"BUZZER"(蜂鳴器控制)
      SET     M5989  ; 指令比對無符合字串條件
      MPP
      FMOV    K0 D10600 K10
3445  LD      M5990  ; SES->EQP上位下達命令觸發自保持
      MPS
      AND     M5901  ; SECS_上位下"START"
      MOVP    D8918 D9075  ; 設備狀態(1Run,2Idle,3Down,4PM)
        [note] "START CMD"
      LD<>    D9075 K1  ; 設備狀態(1Run,2Idle,3Down,4PM)
      AND<>   D9075 K2  ; 設備狀態(1Run,2Idle,3Down,4PM)
      OR      M5974  ; "START"_上位允許放板自保持
      ANB
      ANI     M5941  ; "START"_執行條件判定OK
      SET     M5921  ; "START"_執行條件判定NG
      MPP
      AND     M5901  ; SECS_上位下"START"
      ANI     M5921  ; "START"_執行條件判定NG
      SET     M5941  ; "START"_執行條件判定OK
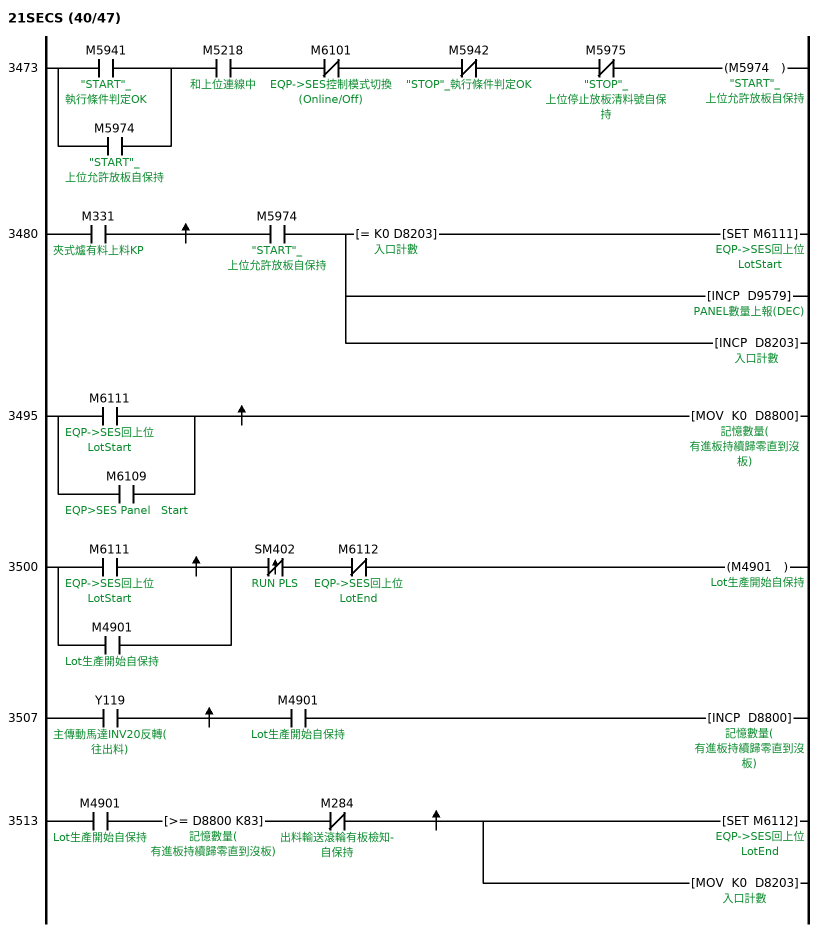
3473  LD      M5941  ; "START"_執行條件判定OK
      OR      M5974  ; "START"_上位允許放板自保持
      AND     M5218  ; 和上位連線中
      ANI     M6101  ; EQP->SES控制模式切換(Online/Off)
      ANI     M5942  ; "STOP"_執行條件判定OK
      ANI     M5975  ; "STOP"_ 上位停止放板清料號自保持
      OUT     M5974  ; "START"_上位允許放板自保持
3480  LD      M331  ; 夾式爐有料上料KP
      MEP
      AND     M5974  ; "START"_上位允許放板自保持
      MPS
      AND=    K0 D8203  ; 入口計數
      SET     M6111  ; EQP->SES回上位  LotStart
      MPP
      INCP    D9579  ; PANEL數量上報(DEC)
      INCP    D8203
3495  LD      M6111  ; EQP->SES回上位  LotStart
      OR      M6109  ; EQP>SES Panel   Start
      MEP
      MOV     K0 D8800  ; 記憶數量(有進板持續歸零直到沒板)
3500  LD      M6111  ; EQP->SES回上位  LotStart
      MEP
      OR      M4901  ; Lot生產開始自保持
      ANDPI   SM402  ; RUN PLS
      ANI     M6112  ; EQP->SES回上位  LotEnd
      OUT     M4901  ; Lot生產開始自保持
3507  LD      Y119  ; 主傳動馬達INV20反轉(往出料)
      MEP
      AND     M4901  ; Lot生產開始自保持
      INCP    D8800
3513  LD      M4901  ; Lot生產開始自保持
      AND>=   D8800 K83  ; 記憶數量(有進板持續歸零直到沒板)
      ANI     M284  ; 出料輸送滾輪有板檢知-自保持
      MEP
      SET     M6112  ; EQP->SES回上位  LotEnd
      MOV     K0 D8203
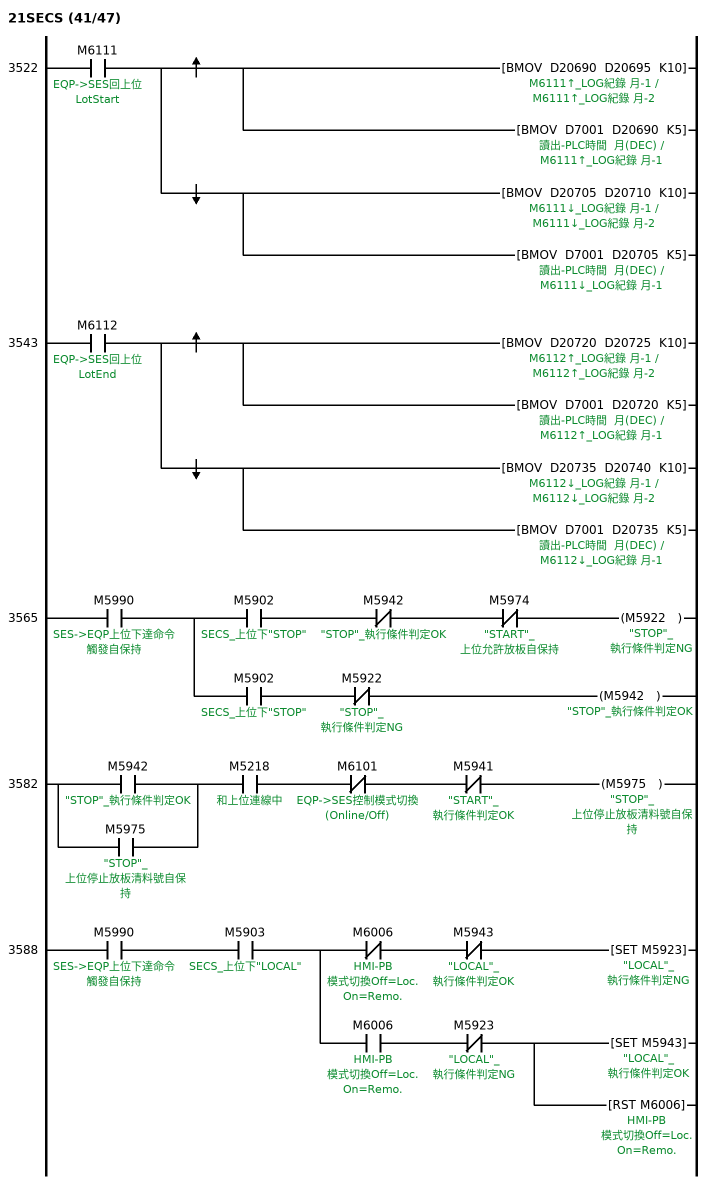
3522  LD      M6111  ; EQP->SES回上位  LotStart
      MPS
      MEP
      BMOV    D20690 D20695 K10  ; M6111↑_LOG紀錄 月-1 / M6111↑_LOG紀錄 月-2
      BMOV    D7001 D20690 K5
      MPP
      MEF
      BMOV    D20705 D20710 K10  ; M6111↓_LOG紀錄 月-1 / M6111↓_LOG紀錄 月-2
      BMOV    D7001 D20705 K5
3543  LD      M6112  ; EQP->SES回上位  LotEnd
      MPS
      MEP
      BMOV    D20720 D20725 K10  ; M6112↑_LOG紀錄 月-1 / M6112↑_LOG紀錄 月-2
      BMOV    D7001 D20720 K5
      MPP
      MEF
      BMOV    D20735 D20740 K10  ; M6112↓_LOG紀錄 月-1 / M6112↓_LOG紀錄 月-2
      BMOV    D7001 D20735 K5
3565  LD      M5990  ; SES->EQP上位下達命令觸發自保持
      MPS
      AND     M5902  ; SECS_上位下"STOP"
      ANI     M5942  ; "STOP"_執行條件判定OK
      ANI     M5974  ; "START"_上位允許放板自保持
      OUT     M5922  ; "STOP"_執行條件判定NG
        [note] "STOP CMD"
      MPP
      AND     M5902  ; SECS_上位下"STOP"
      ANI     M5922  ; "STOP"_執行條件判定NG
      OUT     M5942  ; "STOP"_執行條件判定OK
3582  LD      M5942  ; "STOP"_執行條件判定OK
      OR      M5975  ; "STOP"_ 上位停止放板清料號自保持
      AND     M5218  ; 和上位連線中
      ANI     M6101  ; EQP->SES控制模式切換(Online/Off)
      ANI     M5941  ; "START"_執行條件判定OK
      OUT     M5975  ; "STOP"_ 上位停止放板清料號自保持
3588  LD      M5990  ; SES->EQP上位下達命令觸發自保持
      AND     M5903  ; SECS_上位下"LOCAL"
      MPS
      ANI     M6006  ; HMI-PB  模式切換Off=Loc.On=Remo.
      ANI     M5943  ; "LOCAL"_執行條件判定OK
      SET     M5923  ; "LOCAL"_執行條件判定NG
        [note] "LOCAL CMD"
      MPP
      AND     M6006  ; HMI-PB  模式切換Off=Loc.On=Remo.
      ANI     M5923  ; "LOCAL"_執行條件判定NG
      SET     M5943  ; "LOCAL"_執行條件判定OK
      RST     M6006  ; HMI-PB  模式切換Off=Loc.On=Remo.
